	i1ProTankPumpLPM : INT; (* Byte "n+100, n+101" *)
	i2ProTankPumpHz : INT; (* Byte "n+102, n+103" *)
	i3ProTankBtmUsAPwrPercent : INT; (* Byte "n+104, n+105" *)
	i4ProTankBtmUsBPwrPercent : INT; (* Byte "n+106, n+107" *)
	i5ProTankBtmUsCPwrPercent : INT; (* Byte "n+108, n+109" *)
	i6ProTankSideUsAPwrPercent : INT; (* Byte "n+110, n+111" *)
	i7ProTankSideUsBPwrPercent : INT; (* Byte "n+112, n+113" *)
	i8ProTankBtmUsAkHz : INT; (* Byte "n+114, n+115" *)
	i9ProTankBtmUsBkHz : INT; (* Byte "n+116, n+117" *)
	i10ProTankBtmUsCkHz : INT; (* Byte "n+118, n+119" *)
	i11ProTankSideUsAkHz : INT; (* Byte "n+120, n+121" *)
	i12ProTankSideUsBkHz : INT; (* Byte "n+122, n+123" *)
	i13ProTankBlowerHz : INT; (* Byte "n+124, n+125" *)
	r14ProTankChangeTempDegC : REAL; (*Byte " n+126, n+129" *) (*New*)
	r15SubTankChangeTempDegC :REAL; (*Byte "N+130, n+133" *) (*New*)
	i16SubTankPumpLPM : INT; (*Byte "N+134, n+135" *) (*New*)
	i17SubTankPumpHz : INT; (*Byte "N+136, n+137" *) (*New*)
	i18SlowPullVelocity   : INT;(* Byte "n+154, n+155" *) (*MODIFIED*)
	i19SlowPullDelayTime   : INT;(* Byte "n+154, n+155" *) (*MODIFIED*)


	sReservedInt : STRING(50); (* Byte "n+138~n+199" *)





END_STRUCT
END_TYPE

// ---- DUTs/DS TBD/DS_SubRecipeMemory.TcDUT
TYPE DS_SubRecipeMemory : (*Full Occupied Byte = 400*)
STRUCT
(*BOOL - Start Condition*)
(*	bStCon1EnLowLiquidLevel : BOOL; (* Byte "n" *)
	bStCon2EnRegLiquidLevel : BOOL; (* Byte "n+1" *)
	bStCon3EnLowVacuumLevel : BOOL; (* Byte "n+2" *)
	bStCon4EnRegVacuumLevel : BOOL; (* Byte "n+3" *)
	bStCon5EnLowPressureLevel : BOOL; (* Byte "n+4" *)
	bStCon6EnRegPressureLevel : BOOL; (* Byte "n+5" *)
	bStCon7EnBelowTargetVacuumLevel : BOOL; (* Byte "n+6" *)
	bStCon8EnAboveTargetVacuumLevel : BOOL; (* Byte "n+7" *)
	bStCon9EnBelowTargetPressureLevel : BOOL; (* Byte "n+8" *)
	bStCon10EnAboveTargetPressureLevel : BOOL; (* Byte "n+9" *)
	bStCon11EnBelowTargetProTankTempLevel : BOOL; (* Byte "n+10" *)
	bStCon12EnAboveTargetProTankTempLevel : BOOL; (* Byte "n+11" *)
	bStCon13EnBelowTargetSubTankTempLevel : BOOL; (* Byte "n+12" *)
	bStCon14EnAboveTargetSubTankTempLevel : BOOL; (* Byte "n+13" *)
	bStCon15ExternalActivation : BOOL; (* Byte "n+14" *)
*)
	bStCon1EnProLowLiquidLevel : BOOL; (* Byte "n" *)
	bStCon2EnProRegLiquidLevel : BOOL; (* Byte "n+1" *)
	bStCon3EnProHighLiquidLevel : BOOL; (* Byte "n+1" *)

	bStCon4EnSubLowLiquidLevel : BOOL; (* Byte "n+1" *)
	bStCon5EnSubRegLiquidLevel : BOOL; (* Byte "n+1" *)
	bStCon6EnSubHighLiquidLevel : BOOL; (* Byte "n+1" *)

	bStCon7EnLowVacuumLevel : BOOL; (* Byte "n+2" *)
	bStCon8EnRegVacuumLevel : BOOL; (* Byte "n+3" *)
	bStCon9EnLowPressureLevel : BOOL; (* Byte "n+4" *)
	bStCon10EnRegPressureLevel : BOOL; (* Byte "n+5" *)
	bStCon11EnBelowTargetVacuumLevel : BOOL; (* Byte "n+6" *)
	bStCon12EnAboveTargetVacuumLevel : BOOL; (* Byte "n+7" *)
	bStCon13EnBelowTargetPressureLevel : BOOL; (* Byte "n+8" *)
	bStCon14EnAboveTargetPressureLevel : BOOL; (* Byte "n+9" *)
	bStCon15EnBelowTargetProTankTempLevel : BOOL; (* Byte "n+10" *)
	bStCon16EnAboveTargetProTankTempLevel : BOOL; (* Byte "n+11" *)
	bStCon17EnBelowTargetSubTankTempLevel : BOOL; (* Byte "n+12" *)
	bStCon18EnAboveTargetSubTankTempLevel : BOOL; (* Byte "n+13" *)
	bStCon19ExternalActivation : BOOL; (* Byte "n+14" *)

(*BOOL - Complete Condition*)
	bComCon1EnProLowLiquidLevel : BOOL; (* Byte "n+15" *)
	bComCon2EnProRegLiquidLevel : BOOL; (* Byte "n+16" *)
	bComCon3EnProHighLiquidLevel : BOOL; (* Byte "n+16" *)

	bComCon4EnSubLowLiquidLevel : BOOL; (* Byte "n+16" *)
	bComCon5EnSubRegLiquidLevel : BOOL; (* Byte "n+16" *)
	bComCon6EnSubHighLiquidLevel : BOOL; (* Byte "n+16" *)

	bComCon7EnLowVacuumLevel : BOOL; (* Byte "n+17" *)
	bComCon8EnRegVacuumLevel : BOOL; (* Byte "n+18" *)
	bComCon9EnLowPressureLevel : BOOL; (* Byte "n+19" *)
	bComCon10EnRegPressureLevel : BOOL; (* Byte "n+20" *)
	bComCon11EnBelowTargetVacuumLevel : BOOL; (* Byte "n+21" *)
	bComCon12EnAboveTargetVacuumLevel : BOOL; (* Byte "n+22" *)
	bComCon13EnBelowTargetPressureLevel : BOOL; (* Byte "n+23" *)
	bComCon14EnAboveTargetPressureLevel : BOOL; (* Byte "n+24" *)
	bComCon15EnBelowTargetProTankTempLevel : BOOL; (* Byte "n+25" *)
	bComCon16EnAboveTargetProTankTempLevel : BOOL; (* Byte "n+26" *)
	bComCon17EnBelowTargetSubTankTempLevel : BOOL; (* Byte "n+27" *)
	bComCon18EnAboveTargetSubTankTempLevel : BOOL; (* Byte "n+28" *)
	bComCon19EnExternalActivation : BOOL; (* Byte "n+29" *)
	bComCon20EnProcessTimer : BOOL; (* Byte "n+29" *)

(*BOOL - Instrument Output*)
	bOut1EnProTankPump : BOOL; (* Byte "n+30" *)
	bOut2EnProTankHeater : BOOL; (* Byte "n+31" *)
	bOut3EnProTankBottomUltrasonicA : BOOL; (* Byte "n+32" *)
	bOut4EnProTankBottomUltrasonicB : BOOL; (* Byte "n+33" *)
	bOut5EnProTankBottomUltrasonicC : BOOL; (* Byte "n+34" *)
	bOut6EnProTankSideUltrasonicA : BOOL; (* Byte "n+35" *)
	bOut7EnProTankSideUltrasonicB : BOOL; (* Byte "n+36" *)
	bOut8EnSubTankPump : BOOL; (* Byte "n+37" *)
	bOut9EnSubTankHeater : BOOL; (* Byte "n+38" *)
	bOut10EnBlower : BOOL; (* Byte "n+39" *)
	bOut11EnVacuumPump : BOOL; (* Byte "n+40" *)
	bOut12EnSlowPull : BOOL; (* Byte "n+41" *) (*MODIFIED*)
	bOut13EnInstrument2 : BOOL; (* Byte "n+42" *)
	bOut14EnInstrument3 : BOOL; (* Byte "n+43" *)
	bOut15EnInstrument4 : BOOL; (* Byte "n+44" *)

(*BOOL - Valve Output*)
	bOut1ActValve1 : BOOL; (* Byte "n+45" *)
	bOut2ActValve2 : BOOL; (* Byte "n+46" *)
	bOut3ActValve3 : BOOL; (* Byte "n+47" *)
	bOut4ActValve4 : BOOL; (* Byte "n+48" *)
	bOut5ActValve5 : BOOL; (* Byte "n+49" *)
	bOut6ActValve6 : BOOL; (* Byte "n+50" *)
	bOut7ActValve7 : BOOL; (* Byte "n+51" *)
	bOut8ActValve8 : BOOL; (* Byte "n+52" *)
	bOut9ActValve9 : BOOL; (* Byte "n+53" *)
	bOut10ActValve10 : BOOL; (* Byte "n+54" *)
	bOut11ActValve11 : BOOL; (* Byte "n+55" *)
	bOut12ActValve12 : BOOL; (* Byte "n+56" *)
	bOut13ActValve13 : BOOL; (* Byte "n+57" *)
	bOut14ActValve14 : BOOL; (* Byte "n+58" *)
	bOut15ActValve15 : BOOL; (* Byte "n+59" *)
	bOut16ActValve16 : BOOL; (* Byte "n+60" *)
	bOut17ActValve17 : BOOL; (* Byte "n+61" *)
	bOut18ActValve18 : BOOL; (* Byte "n+62" *)
	bOut19ActValve19 : BOOL; (* Byte "n+63" *)
	bOut20ActValve20 : BOOL; (* Byte "n+64" *)


(*BOOL - Instrument Output*) (*New*)
	bOut16EnProTankChangeTemperature : BOOL; (* Byte "n+65" *) (*New*)
	bOut17EnSubTankChangeTemperature : BOOL; (* Byte "n+66" *) (*New*)


	sReservedBool : STRING(50); (* Byte "n+67~n+99" *)


(*INT - Start Condition*)

	iStCon1TargetVacuumLevel : INT; (* Byte "n+100, n+101" *)
	iStCon2TargetPressureLevel : INT; (* Byte "n+102, n+103" *)
	iStCon3TargetProTankTempLevel : INT; (* Byte "n+104, n+105" *)
	iStCon4TargetSubTankTempLevel : INT; (* Byte "n+106, n+107" *)

(*INT - Complete Condition*)

	iComCon1TargetVacuumLevel : INT; (* Byte "n+108, n+109" *)
	iComCon2TargetPressureLevel : INT; (* Byte "n+110, n+111" *)
	iComCon3TargetProTankTempLevel : INT; (* Byte "n+112, n+113" *)
	iComCon4TargetSubTankTempLevel : INT; (* Byte "n+114, n+115" *)
	iComCon5ProcessTimer : INT; (* Byte "n+116, n+117" *)

(*INT - Power/Flow Control*)
	iOut1ProTankPumpLPM : INT; (* Byte "n+118, n+119" *)
	iOut2ProTankPumpHz : INT; (* Byte "n+120, n+121" *)
	iOut3ProTankBtmUsAPwrPercent : INT; (* Byte "n+122, n+123" *)
	iOut4ProTankBtmUsBPwrPercent : INT; (* Byte "n+124, n+125" *)
	iOut5ProTankBtmUsCPwrPercent : INT; (* Byte "n+126, n+127" *)
	iOut6ProTankSideUsAPwrPercent : INT; (* Byte "n+128, n+129" *)
	iOut7ProTankSideUsBPwrPercent : INT; (* Byte "n+130, n+131" *)
	iOut8ProTankBtmUsAkHz : INT; (* Byte "n+132, n+133" *)
	iOut9ProTankBtmUsBkHz : INT; (* Byte "n+134, n+135" *)
	iOut10ProTankBtmUsCkHz : INT; (* Byte "n+136, n+137" *)
	iOut11ProTankSideUsAkHz : INT; (* Byte "n+138, n+139" *)
	iOut12ProTankSideUsBkHz : INT; (* Byte "n+140, n+141" *)
	iOut13ProTankBlowerHz : INT;(* Byte "n+142, n+143" *)

	rOut14ProTankChangeTemperatureDegC  : REAL;(* Byte "n+144, n+147" *) (*New*)
	rOut15SubTankChangeTemperatureDegC  : REAL;(* Byte "n+148, n+151" *) (*New*)
	iOut16SubTankPumpLPM   : INT;(* Byte "n+152, n+153" *) (*New*)
	iOut17SubTankPumpHz   : INT;(* Byte "n+154, n+155" *) (*New*)

	iOut18SlowPullVelocity   : INT;(* Byte "n+154, n+155" *) (*MODIFIED*)
	iOut19SlowPullDelayTime   : INT;(* Byte "n+154, n+155" *) (*MODIFIED*)



	sReservedInt : STRING(50); (* Byte "n+156~n+159" *)


(*LREAL - Standby*)
	lrLREALReserved1 : LREAL; (* Byte "n+160~n+167" *)
	lrLREALReserved2 : LREAL; (* Byte "n+168~n+175" *)
	sReservedLreal : STRING(50); (* Byte "n+176~n+199" *)


(*STRING - Standby*)
	sStringReserved1 : STRING(50); (* Byte "n+200 ~ n+299" *)
	sStringReserved2 : STRING(50); (* Byte "n+300 ~ n+399" *)







END_STRUCT
END_TYPE

// ---- DUTs/DS TBD/DS_TimeTrackerInput.TcDUT
TYPE DS_TimeTrackerInput :
STRUCT
(* from DSA1_PnpSequenceMemory*)

(*	bTimeTrackerEn : BOOL;*)
	iTimeTrackerProductRecipeNo : INT;
(*	iTimeTrackerStepNo : INT; (*Byte "n+110, n+111" *) (***************NEW******************)*)

	ARiCallArmNo : ARRAY [0..iProductRecipeStepArrayQty] OF INT; (* Byte "n+100~n+161" *)

	ARiPickStationNo : ARRAY [0..iProductRecipeStepArrayQty] OF INT; (* Byte "n+162~n+223" *)
	ARiTransferStationNo : ARRAY [0..iProductRecipeStepArrayQty] OF INT; (* Byte "n+224~n+285" *)

	ARiStnSeqRepNo : ARRAY [0..iProductRecipeStepArrayQty] OF INT; (* Byte "n+596~n+657" *)

END_STRUCT

END_TYPE

// ---- DUTs/DS TBD/DS_WeberEnclosure.TcDUT
TYPE DS_WeberEnclosure :
STRUCT
	DSWeberGenerator : ARRAY [1..iUSGeneratorQty] OF DS_WeberGenerator;
END_STRUCT
END_TYPE

// ---- DUTs/DS TBD/DS_WeberGenerator.TcDUT
TYPE DS_WeberGenerator :
STRUCT
	IN_bUltrasonicStartEn : BOOL;
	IN_bMultiFreqEn :  BOOL;
	IN_iFreqSetPoint :  INT; (* 40/80/120 or 25/50*)
	IN_iTargetPowerPercentSetPoint :  INT; (* 0-100%*)
	IN_lrPowerToAnalogRatio : LREAL; (*Normally for 0-100% is 327.67*)
	IN_lrAnalogInputFineTuneRatio :  LREAL; (*Normally 1, use lower than 1 (example: 0.97) if set to 100% the actual output is greater, use higher than 1 meant the actual output is lesser when you set 100% *)
	IN_lrAnalogOutputFineTuneRatio :  LREAL; (*Normally 1, use lower than 1 (example: 0.97) if set to 100% the actual output is greater, use higher than 1 meant the actual output is lesser when you set 100% *)

	DSWeberMulFreqSwitching : DS_WeberMulFreqSwitching;

	OUT_bUltrasonicOnOff :  BOOL;
	OUT_iActualPowerPercentDisplay :  INT; (*Display 0 - 100%*)
	OUT_bFreqSetPointError :  BOOL;

	IN_iPowerAnalogInput  :  INT; (*Link to Terminal*)
	OUT_iPowerAnalogOutput  :  INT; (*Link to Terminal*)

END_STRUCT
END_TYPE

// ---- DUTs/DS TBD/DS_WeberMulFreqSwitching.TcDUT
TYPE DS_WeberMulFreqSwitching :
STRUCT
	bFreqSwitchingPB_TS : BOOL;
	bFreqRange4080120En : BOOL;
	bFreqRange2550En : BOOL;
	bDisableMultiFreq80kHz : BOOL;
	bDisableMultiFreq40kHz : BOOL;
	iFreqOutput_TS : INT;
END_STRUCT
END_TYPE

// ---- DUTs/DS TBD/DS_XMLRW.TcDUT
TYPE DS_XMLRW :
STRUCT

	sMachineOnTime_JKS	: STRING(99);

END_STRUCT
END_TYPE

// ---- DUTs/DS TBD/DS_XML_InputOutput.TcDUT
TYPE DS_XML_InputOutput :
STRUCT

(*	var1									: ARRAY [1..iStnQty] OF BOOL;
	ARrStnTempSV_map					: ARRAY [1..iStnQty] OF REAL;
	ARrStnTempPV_map					: ARRAY [1..iStnQty] OF REAL;
	ARrStnTempHALsv_map				: ARRAY [1..iStnQty] OF REAL;
	ARrStnTempRDYsv_map				: ARRAY [1..iStnQty] OF REAL;
	ARrStnTempHYSsv_map				: ARRAY [1..iStnQty] OF REAL;
	ARrStnTemp1stLimitSv_map			: ARRAY [1..iStnQty] OF REAL;
	ARiStnPreparationTempSv_map		: ARRAY [1..iStnQty] OF INT;

	ARrStnSubTankTempSV_map			: ARRAY [1..iStnQty] OF REAL;
	ARrStnSubTankTempPV_map			: ARRAY [1..iStnQty] OF REAL;
	ARrStnSubTankTempHALsv_map		: ARRAY [1..iStnQty] OF REAL;
	ARrStnSubTankTempRDYsv_map		: ARRAY [1..iStnQty] OF REAL;
	ARrStnSubTankTempHYSsv_map		: ARRAY [1..iStnQty] OF REAL;
	ARrStnSubTankTemp1stLimitSv_map	: ARRAY [1..iStnQty] OF REAL;
	ARiStnSubTankPreparationTempSv_map: ARRAY [1..iStnQty] OF INT;


	ARiStnDippingTimeSV_map			: ARRAY [1..iStnQty] OF INT;
	ARiStnToleranceTimeSV_map			: ARRAY [0..iStnQty] OF INT;
	ARiStnTopUpDelayOffTimeSV_map		: ARRAY [1..iStnQty] OF INT;
*)
	ARrStnConductivityPV_map 			: ARRAY [1..iStnQty] OF REAL;
	ARrStnConductivity1stLimitSv_map		: ARRAY [1..iStnQty] OF REAL;
	ARrStnConductivity2ndLimitSv_map		: ARRAY [1..iStnQty] OF REAL;
(*
	ARrStnPhPV_map						: ARRAY [1..iStnQty] OF REAL;
	ARrStnLowPHSv_map					: ARRAY [1..iStnQty] OF REAL;
	ARrStnHighPHSv_map					: ARRAY [1..iStnQty] OF REAL;

	ARrStnFilterPressurePV_map 			: ARRAY [1..iStnQty] OF REAL;
	ARrStnLowFilterPressureSv_map		: ARRAY [1..iStnQty] OF REAL;
	ARrStnHighFilterPressureSv_map		: ARRAY [1..iStnQty] OF REAL;
*)
END_STRUCT
END_TYPE

// ---- DUTs/DS TBD/En_LogFileType.TcDUT
TYPE En_LogFileType :
(
	CSV:=1,
	TXT:=2
);
END_TYPE

// ---- DUTs/DS TBD/En_TimeInterval.TcDUT
TYPE En_TimeInterval :
(
	Interval_1s:=12,
	Interval_5s:=13,
	Interval_10s:=0,
	Interval_20s:=1,
	Interval_30s:=2,
	Interval_1min:=3,
	Interval_2min:=4,
	Interval_5min:=5,
	Interval_10min:=6,
	Interval_15min:=7,
	Interval_20min:=8,
	Interval_30min:=9,
	Interval_1h:=10,
	Interval_2h:=11

);
END_TYPE

// ---- DUTs/DS Twincat 3/Barcode/DS_SerialCommunication.TcDUT
TYPE DS_SerialCommunication :
STRUCT
	// Config
	SerialCfg 				: ComSerialConfig;
	PortOpened 				: BOOL;     (* Indicates if selected serial port is opened *)
    SerialConnectError      : BOOL;     (* 'TRUE' if an error occurred *)
    ErrorID    				: UDINT;    (* Displays the error code; 0 = no error *)
    Busy       				: BOOL;     (* 'TRUE' if internal ADS communication is busy *)
    TxBufCount 				: UDINT;    (* number of bytes in internal Tx buffer *)
    RxBufCount 				: UDINT;    (* number of bytes in internal Rx buffer *)	
    Error 					: BOOL;
	RxTimeout 				: BOOL;
	StringReceived 			: BOOL;
	TxBuffer				: ComBuffer;
	RxBuffer				: ComBuffer;

	// Send String Input
	sSendString 			: STRING;
	bSendStringBusy 		: BOOL;
	SendStringError 		: ComError_t;
	
	// Receive String Input//
	sReceivedString 		: STRING;
	bStringReceived			: BOOL;
	ReceivedStringError 	: ComError_t;
	bReceivedStringBusy 	: BOOL;
	bReceivedStringTimeout	: BOOL;
	bReceivedStringReset	: BOOL;	
	sRSPrefix 				: STRING;
    sRSSuffix 				: STRING;
	
END_STRUCT
END_TYPE

// ---- DUTs/DS Twincat 3/CSV/DS_CsvErrorLog.TcDUT
TYPE DS_CsvErrorLog EXTENDS DS_CsvLog :
STRUCT
	udiErrorId	: UDINT;
	iCaseid		: INT;
END_STRUCT
END_TYPE

// ---- DUTs/DS Twincat 3/CSV/DS_CsvLog.TcDUT
TYPE DS_CsvLog :
STRUCT
		eLogAction			: E_CsvActionType; 
		sPathAndFilename	: STRING(255);
		sLogString			: STRING(255);
END_STRUCT
END_TYPE

// ---- DUTs/DS Twincat 3/CSV/DS_CsvReport.TcDUT
TYPE DS_CsvReport :
STRUCT
	
	ARsHeadlineTitle			: ARRAY [1..100] OF STRING;		// Please consider to replace the name on next project
	ARsHeadlineData				: ARRAY [1..100] OF STRING;	                		
	ARsLogUnit					: ARRAY [1..100] OF STRING;
	ARsLogTitle					: ARRAY [1..100] OF STRING;
	AR2sLogData					: ARRAY [1..100]OF ARRAY [1..C_iCsvDataBlockQty] OF STRING;

	iNumOfData_HeadlineTitle 	: INT := 50;
	iNumOfData_HeadlineData		: INT := 50;
	iNumOfData_LogUnit			: INT := 50;
	iNumOfData_LogTitle			: INT := 50;
	iNumOfData_LogData			: INT := 50;

	ARsLogTitle_EventLog 			: ARRAY [1..C_iCsvDataBlockQty] OF STRING;
	ARsLogData_EventLog 			: ARRAY [1..C_iCsvDataBlockQty] OF STRING;

	iNumOfData_LogTitle_EventLog 	: INT := 10;
	iNumOfData_LogData_EventLog 	: INT := 10;
	
	ARsLogBuffer		: ARRAY [1..C_udiCsvBufferByteQty] OF BYTE; 
	
END_STRUCT
END_TYPE

// ---- DUTs/DS Twincat 3/CSV/E_CsvActionType.TcDUT
{attribute 'Tc2GvlVarNames'}
{attribute 'strict'}
{attribute 'to_String'}
TYPE E_CsvActionType :
(
	eCsvNewFile_CarrierReport 	:= 1,
	eCsvLogData_CarrierReport	:= 2,
	eCsvGenerate_CarrierReport	:= 3,
	eCsvNewFile_EventLog 		:= 4,
	eCsvLogData_EventLog		:= 5,
	eCsvGenerate_EventLog		:= 6
	
);
END_TYPE

// ---- DUTs/DS Twincat 3/DS_HMI_MappingVariable.TcDUT
TYPE DS_HMI_MappingVariable :
STRUCT
	
//PushButton

bProTankHeater_PB				:BOOL;
bProTankPump_PB				    :Bool;
bProTankUsSide_PB				:Bool;
bProTankUsBtm_PB				:Bool;
bProTankUsFreqChangeBit1_PB	    :Bool;
bProTankUsFreqChangeBit2_PB     :Bool;
bProTankVacuumPump_PB			:Bool;
bProTankAgitationMotor_PB		:BOOL;
bProTankBlower_PB				:BOOL;
bDosingPump_PB				    :BOOL;
bLdConveyorMotor01_PB			:BOOL;
bLdConveyorMotor02_PB			:BOOL;
bLdConveyorMotor03_PB			:BOOL;
bLdConveyorMotor04_PB			:BOOL;
bValve01_PB					    :BOOL;
bValve02_PB					    :Bool;
bValve03_PB					    :Bool;
bValve04_PB					    :Bool;
bValve05_PB					    :BOOL;
bExhaustBlower_PB				:BOOL;
bStnRotationRotaryBarrel_PB		:BOOL;
bRobotRotationRotaryBarrel_PB   :BOOL;
bGeneralIncValve01_PB 			:BOOL;
bGeneralIncValve02_PB 			:BOOL;
bFFU01_PB				 		:BOOL;
bFFU02_PB				 		:BOOL;




//Indicator
bProTankHeater_IND				:BOOL;
bProTankPump_IND	  			:BOOL;
bProTankUsSide_IND				:BOOL;
bProTankUsBtm_IND				:BOOL;
bProTankUsFreqChangeBit1_IND	:BOOL;
bProTankUsFreqChangeBit2_IND    :BOOL;
bProTankVacuumPump_IND			:BOOL;
bProTankAgitationMotor_IND		:BOOL;
bProTankBlower_IND				:BOOL;
bDosingPump_IND	    			:BOOL;
bLdConveyorMotor01_IND			:BOOL;
bLdConveyorMotor02_IND			:BOOL;
bLdConveyorMotor03_IND			:BOOL;
bLdConveyorMotor04_IND			:BOOL;
bValve01_IND			  		:BOOL;
bValve02_IND			  		:BOOL;
bValve03_IND			  		:BOOL;
bValve04_IND			  		:BOOL;
bValve05_IND			  		:BOOL;
bExhaustBlower_IND				:BOOL;
bStnRotationRotaryBarrel_IND	:BOOL;
bRobotRotationRotaryBarrel_IND  :BOOL;
bGeneralIncValve01_IND 			:BOOL;
bGeneralIncValve02_IND 			:BOOL;


bProcessTankMinLevel_IND		:BOOL;
bProcessTankRegLevel_IND		:BOOL;
bProcessTankTopupLevel_IND		:BOOL;

bSubTankMinLevel_IND			:BOOL;
bSubTankRegLevel_IND			:BOOL;
bSubTankMaxLevel_IND			:BOOL;
bSubTankTopupLevel_IND			:BOOL;

bOverflowMinLevel_IND			:BOOL;
bOverflowRegLevel_IND			:BOOL;
bOverflowMaxLevel_IND			:BOOL;

bLdFeedSensor_IND				:BOOL;
bLdIndex1Sensor_IND				:BOOL;
bLdIndex2Sensor_IND				:BOOL;
bLdIndex3Sensor_IND				:BOOL;
bLdIndex4Sensor_IND				:BOOL;
bLdPickSensor_IND				:BOOL;

bUldFeedSensor_IND				:BOOL;
bUldIndex1Sensor_IND			:BOOL;
bUldIndex2Sensor_IND			:BOOL;
bUldIndex3Sensor_IND			:BOOL;
bUldIndex4Sensor_IND			:BOOL;
bUldPickSensor_IND				:BOOL;

bFFU01_IND				 		:BOOL;
bFFU02_IND				 		:BOOL;




END_STRUCT
END_TYPE

// ---- DUTs/DS Twincat 3/DS_LocalSystemTime.TcDUT
TYPE DS_LocalSystemTime :
STRUCT

dtCurrentDateTime			: DT; 		  // Newly Added DT#2023-02-20-15:49:44
sCurrentDateTime			: STRING(30); // Newly Added 2023-02-20-15:49:44
sCurrentDate_General		: STRING(255); // Newly Added YYYYMMDD
sCurrentTime24Hr_General	: STRING(50); // Newly Added HH:MM:SS	
sCurrentDT24Hr_General		: STRING(50);
sCurrentDT12Hr				: STRING(50);
sCurrentDT24Hr				: STRING(50);
sDayOfWeek					: STRING(10);
sYear						: STRING(10);
sMonth						: STRING(10);
sDay						: STRING(10);
s24Hour						: STRING(10);
s12Hour						: STRING(10);
sMin						: STRING(10);
sSec						: STRING(10);
s12HrSign					: STRING(10);

END_STRUCT
END_TYPE

// ---- DUTs/DS Twincat 3/DS_XML_Persistent_Analog.TcDUT
TYPE DS_XML_Persistent_Analog :
STRUCT
	(* xxxxxxxxxxxxxxxxxxxxxxxxxxxxxxxx Temperature Cltr xxxxxxxxxxxxxxxxxxxxxxxxxxxxxxxx*)
(*========================================================================*)

	ARfbStnTempControl									: ARRAY [1..iStnQty] OF fbV2_TempControl;

	ARrAnalogInputFineTuneRatio							: ARRAY [1..iStnQty] OF REAL;

	ARrStnTempHYSsv										: ARRAY [1..iStnQty] OF REAL;
	ARrStnTempHALsv										: ARRAY [1..iStnQty] OF REAL;
	ARrStnTempSV										: ARRAY [1..iStnQty] OF REAL;
	ARrStnTempRDYsv										: ARRAY [1..iStnQty] OF REAL;
	ARrStnTemp1stLimitSv								: ARRAY [1..iStnQty] OF REAL;
	ARrStnTemp2ndLimitSv								: ARRAY [1..iStnQty] OF REAL;
	ARiStnPreparationTempSv								: ARRAY [1..iStnQty] OF INT;
	
	fbChillerSystemTempControl							: fbV2_TempControl;
	
	rChillerSystemAnalogInputFineTuneRatio				: REAL;

	rChillerSystemTempHYSsv								: REAL;
	rChillerSystemTempHALsv								: REAL;
	rChillerSystemTempSV								: REAL;
	rChillerSystemTempRDYsv								: REAL;
	rChillerSystemTemp1stLimitSv						: REAL;
	rChillerSystemTemp2ndLimitSv						: REAL;
	iChillerSystemPreparationTempSv						: INT;

	ARrStnChillerValueTempSetpoint						: ARRAY [1..iStnQty] OF REAL;
	
(*****Temperature Changed Based on Recipe Ctrl *****)

	fbTemperatureParaRecipe								: fbV3_TemperatureParaRecipe;

	DSTempCtrlParameter_Min 							: DSV3_TempCtrlParameter;
	DSTempCtrlParameter_Max 							: DSV3_TempCtrlParameter;

	HMI_DSTempCtrlParameter_Input 						: DSV3_TempCtrlParameter;

(* xxxxxxxxxxxxxxxxxxxxxxxxxxxxxxxx Conductivity Cltr xxxxxxxxxxxxxxxxxxxxxxxxxxxxxxxx*)
(*========================================================================*)

	ARfbStnConductivity 								: ARRAY [1..iStnQty] OF fbRawRatioConversionReal;

	ARrStnLowConductivitySv								: ARRAY [1..iStnQty] OF REAL;
	ARrStnHighConductivitySv							: ARRAY [1..iStnQty] OF REAL;
	ARrStnConductivity1stLimitSv						: ARRAY [1..iStnQty] OF REAL;
	ARrStnConductivity2ndLimitSv						: ARRAY [1..iStnQty] OF REAL;

	bStnConductivityMaxLimitReach						: ARRAY [1..iStnQty] OF BOOL;
	ARsConductivityMsgStatus							: ARRAY [1..iStnQty] OF STRING;

(* xxxxxxxxxxxxxxxxxxxxxxxxxxxxxxxx Filter Pressure Cltr xxxxxxxxxxxxxxxxxxxxxxxxxxxxxxxx*)
(*========================================================================*)

	ARfbStnFilterPressure 								: ARRAY [1..iStnQty] OF fbRawRatioConversionReal;
                                                    
	ARrStnLowFilterPressureSv							: ARRAY [1..iStnQty] OF REAL;
	ARrStnHighFilterPressureSv							: ARRAY [1..iStnQty] OF REAL;
	ARrStnFilterPressure1stLimitSv						: ARRAY [1..iStnQty] OF REAL;
	ARrStnFilterPressure2ndLimitSv						: ARRAY [1..iStnQty] OF REAL;
                                                    
	ARfbIncFilterPressure								: ARRAY [1..iStnQty] OF fbRawRatioConversionReal;
	ARrIncLowFilterPressureSv							: ARRAY [1..iStnQty] OF REAL;
	ARrIncHighFilterPressureSv							: ARRAY [1..iStnQty] OF REAL;
	ARrIncFilterPressure1stLimitSv						: ARRAY [1..iStnQty] OF REAL;
	ARrIncFilterPressure2ndLimitSv						: ARRAY [1..iStnQty] OF REAL;


(* xxxxxxxxxxxxxxxxxxxxxxxxxxxx Clangsonic Ultrasonic Cltr xxxxxxxxxxxxxxxxxxxxxxxxxxxx*)
(*========================================================================*)

	DSClangGenerator 									: ARRAY [1..iUSGeneratorQty] OF DS_ClangsonicGenerator;
	DSClangGenerator2 									: ARRAY [1..iUSGeneratorQty] OF DS_ClangsonicGenerator;
	iClangStepDelaySVns									: INT := 50;
	iClangStepDelaySVns2								: INT := 50;

	iClangTolerance										: INT;
	iUSTolerance										: INT;
	ARlrUsMaxData_Watt									: ARRAY [1..12] OF LREAL;

	DSClangsonicGenerator 								: DSV2_ClangsonicGenerator;
	DSClangsonicGenerator2 								: DSV2_ClangsonicGenerator;

	
(* xxxxxxxxxxxxxxxxxxxxxxxxxxx Modbus Cltr xxxxxxxxxxxxxxxxxxxxxxxxxxx*)
(*========================================================================*)
	DSV2ModbusControl									: DSV2_ModbusControl;
	DSV2ModbusControl2 									: DSV2_ModbusControl;
	
	IStepDelaySVns										: INT := 50;
	IStepDelaySVns2										: INT := 50;


END_STRUCT
END_TYPE

// ---- DUTs/DS Twincat 3/DS_XML_Persistent_Arm.TcDUT
TYPE DS_XML_Persistent_Arm :
STRUCT
	(* xxxxxxxxxxxxxxxxxxxxxxxxxxxxxxxxxxx  Station Info xxxxxxxxxxxxxxxxxxxxxxxxxxxxxxxxxxx*)
(*========================================================================*)

	bEnableCallArmNo 						: BOOL;
	iCallArmNo 								: INT;
	ARiVertArmPosOffset 					: ARRAY [0..iArmQty] OF INT;

	bAgitationEn							: BOOL;
	bArm2AgitationEn						: BOOL;
(* xxxxxxxxxxxxxxxxxxxxxxxxxxx  Display Product Description xxxxxxxxxxxxxxxxxxxxxxxxxxx*)
(*========================================================================*)

	ARsProductRecipeDescription				: ARRAY [0..iProductRecipeArrayQty] OF STRING(50);
	DSHmiStationDisplayInfo 				: ARRAY [1..iStnQty] OF DS_HMIStationDisplayInfo;

	ARbStnSeqRepNoVisible					: ARRAY [0..iProductRecipeStepArrayQty] OF BOOL;
	ARsStnProcessStatus 					: ARRAY [0..iStnQty] OF STRING;

(* xxxxxxxxxxxxxxxxxxxxxx  Arm PnP Sequence Memory Description xxxxxxxxxxxxxxxxxxxxxx*)
(*========================================================================*)

	DSA1fbPnpSequenceMemoryCall 			: DSV2_A1_fbPnpSequenceMemoryCall;
	DSA1fbPnpSequenceMemoryStore 			: DSV2_A1_fbPnpSequenceMemoryStore;
	DSA21UpDownPatternCall 					: DSA21_UpDownPatternCall;
	DSA21UpDownPatternStore 				: DSA21_UpDownPatternStore;
	DSA31ArmSpeedProfileCall 				: DSA31_ArmSpeedProfileCall;
	DSA31ArmSpeedProfileStore 				: DSA31_ArmSpeedProfileStore;

(* xxxxxxxxxxxxxxxxxxxxxxxxxxxxx Admin Arm Setting xxxxxxxxxxxxxxxxxxxxxxxxxxxxxxxxxxxxxxx*)
(*========================================================================*)

	DSHomingSetting 						: DS_HomingSetting;

	ARDSArmCtrl 							: ARRAY [0..iArmQty] OF DSV2_ArmPosition;
	(*1 = Stn, 2 = Id, 3 = Uld*)
	(*1 = Up, 2 = SPSlanted, 3 = Regular(*midtop*), 4 = AgitationUp, 5 = AgitationDown, 6 = Down, 7 = Unhook, 8 = Hook, 9 = SlantedLeft, 10 = SlantedRight
		,11 = lifter up, 12 = lifter = down*)

(* xxxxxxxxxxxxxxxxxxxxx  4 Step Arm Movement - Auto/Manual Used xxxxxxxxxxxxxxxxxxxxxxxxxx*)
(*==============================================================================*)

	DS4StepsMovement 						: DS_SA_Movement;
	DSManual4StepsMovement					: DS_SA_Movement;


(* xxxxxxxxxxxxxxxxxxxxxxxxxxx Arm 1 Vert / Horz Velo,Acc,Dcc xxxxxxxxxxxxxxxxxxxxxxxxxxx*)
(*========================================================================*)

	ARlrArmVertFix_PosCfmTolerance			: ARRAY [0..iArmQty] OF LREAL;
	ARlrArmVertFix_2ndSpdRange				: ARRAY [0..iArmQty] OF LREAL;

	ARlrArmHorzFix_PosCfmTolerance			: ARRAY [0..iArmQty] OF LREAL;
	ARlrArmHorzFix_2ndSpdRange				: ARRAY [0..iArmQty] OF LREAL;

(* xxxxxxxxxxxxxxxxxxxxxxxxxxxxxxx Jog Control Variable xxxxxxxxxxxxxxxxxxxxxxxxxxxxxxxxxxxxx*)
(*============================================================================*)

	ARrArmVertJogPercent					: ARRAY [1..iArmQty] OF REAL;
	ARrArmVertJogAcc						: ARRAY [1..iArmQty] OF REAL;
	ARrArmVertJogDcc						: ARRAY [1..iArmQty] OF REAL;

	ARrArmHorzJogPercent					: ARRAY [1..iArmQty] OF REAL;
	ARrArmHorzJogAcc						: ARRAY [1..iArmQty] OF REAL;
	ARrArmHorzJogDcc						: ARRAY [1..iArmQty] OF REAL;

	ARlrArmSlowPullJogVelo					: ARRAY [1..iArmSlowPullQty] OF LREAL;
	ARlrArmSlowPullJogAcc					: ARRAY [1..iArmSlowPullQty] OF LREAL;
	ARlrArmSlowPullJogDcc					: ARRAY [1..iArmSlowPullQty] OF LREAL;

(* xxxxxxxxxxxxxxxxxxxxxxxxxxxxxxxxxxxx Homing Variable xxxxxxxxxxxxxxxxxxxxxxxxxxxxxxxxxxxx*)
(*============================================================================*)

	ARrVertHomeDccDelayTimeSec				: ARRAY [0..iArmQty] OF REAL;
	ARrHorzHomeDccDelayTimeSec				: ARRAY [0..iArmQty] OF REAL;

	ARrArmVertHome1stPercent				: ARRAY [0..iArmQty] OF REAL;
	ARrArmVertHome1stPercentAcc				: ARRAY [0..iArmQty] OF REAL;
	ARrArmVertHome1stPercentDcc				: ARRAY [0..iArmQty] OF REAL;

	ARrArmVertHome2ndPercent				: ARRAY [0..iArmQty] OF REAL;
	ARrArmVertHome2ndPercentAcc				: ARRAY [0..iArmQty] OF REAL;
	ARrArmVertHome2ndPercentDcc				: ARRAY [0..iArmQty] OF REAL;

	ARrArmHorzHome1stPercent				: ARRAY [0..iArmQty] OF REAL;
	ARrArmHorzHome1stPercentAcc				: ARRAY [0..iArmQty] OF REAL;
	ARrArmHorzHome1stPercentDcc				: ARRAY [0..iArmQty] OF REAL;

	ARrArmHorzHome2ndPercent				: ARRAY [0..iArmQty] OF REAL;
	ARrArmHorzHome2ndPercentAcc				: ARRAY [0..iArmQty] OF REAL;
	ARrArmHorzHome2ndPercentDcc				: ARRAY [0..iArmQty] OF REAL;

(* xxxxxxxxxxxxxxxxxxxxxxxxxxxxxxxxx ArmHorzZoneConfirm xxxxxxxxxxxxxxxxxxxxxxxxxxxxxxxxx*)
(*============================================================================*)

	ARlrArmHorzStartPoint 					: ARRAY [0..iArmQty] OF LREAL;
	ARlrArmHorzEndPoint 					: ARRAY [0..iArmQty] OF LREAL;

	ARiArmCurrentHorzZoneNo 				: ARRAY [0..iArmQty] OF INT;
	ARbArmInvalidListingErr					: ARRAY [0..iArmQty] OF BOOL;

	ARlrLdHorzCentrePoint 					: ARRAY [0..iLdStnQty] OF LREAL;
	ARlrStnHorzCentrePoint 					: ARRAY [0..iStnQty] OF LREAL;
	ARlrUldHorzCentrePoint 					: ARRAY [0..iUldStnQty] OF LREAL;

	ARbLdHorzZoneConfirm 					: ARRAY [0..iLdStnQty] OF BOOL;
	ARbArm1HorzStnZoneConfirm 				: ARRAY [1..iStnQty] OF BOOL;
	ARbUldHorzZoneConfirm 					: ARRAY [0..iUldStnQty] OF BOOL;

	ARiArm1HorzListing 						: ARRAY [1..50] OF INT;


(* xxxxxxxxxxxxxxxxxxxxxxxxxxxxxxx Pos Num xxxxxxxxxxxxxxxxxxxxxxxxxxxxxxx*)
(*=========================Pos num============================*)

	ARrVertPos_In_TargetSpdHz				: ARRAY [0..iArmQty] OF REAL;
	ARrVertPos_In_2ndSpdHz					: ARRAY [0..iArmQty] OF REAL;

	ARrHorzPos_In_TargetSpdHz				: ARRAY [0..iArmQty] OF REAL;
	ARrHorzPos_In_2ndSpdHz					: ARRAY [0..iArmQty] OF REAL;

(*=========================Arm Servo Ctrl============================*)

	ARlrVertPos_In_HighSpeed 				: ARRAY [1..iArmQty] OF LREAL;
	ARlrVertPos_In_Acc						: ARRAY [1..iArmQty] OF LREAL;
	ARlrVertPos_In_Dcc						: ARRAY [1..iArmQty] OF LREAL;

	ARlrHorzPos_In_HighSpeed 				: ARRAY [1..iArmQty] OF LREAL;
	ARlrHorzPos_In_Acc						: ARRAY [1..iArmQty] OF LREAL;
	ARlrHorzPos_In_Dcc						: ARRAY [1..iArmQty] OF LREAL;

(* xxxxxxxxxxxxxxxxxxxxxxxxxxxxx Arm Move Variable xxxxxxxxxxxxxxxxxxxxxxxxxxxxxxxxxxxxxx*)
(*============================================================================*)

	DS_ArmLifterPosition					: DS_ArmPnPInOut;

	DSArm1VertConfig						: DS_Servo ;
	DSArm1HorzConfig						: DS_Servo ;

	DSArm2VertConfig						: DS_Servo ;
	DSArm2HorzConfig						: DS_Servo ;

(* xxxxxxxxxxxxxxxxxxxxxxxxxxxxx Generate Arm Pick Transfer Bit xxxxxxxxxxxxxxxxxxxxxxxxxxxxx*)
(*============================================================================*)

	bArmPickLd 								: BOOL;
	bArmPickUld 							: BOOL;
	ARbArmPickStn 							: ARRAY [1..iStnQty] OF BOOL;
	bArmTransferLd 							: BOOL;
	bArmTransferUld 						: BOOL;
	ARbArmTransferStn 						: ARRAY [1..iStnQty] OF BOOL;

(* xxxxxxxxxxxxxxxxxxxxxxxxxxxxx HMI Simulate Arm Movement xxxxxxxxxxxxxxxxxxxxxxxxxxxxx*)
(*============================================================================*)

	lrAngleRatio 							: LREAL;
	bHMIArmSimulateEN 						: BOOL;
	iInterval_ms 							: INT;
	lrMaxSimulateNo 						: LREAL;

	lrSimulateHorzXPos						: LREAL;
	lrSimulateVertYPos						: LREAL;

(* xxxxxxxxxxxxxxxxxxxxxxxxxxxxxxxxxx PnP control variable xxxxxxxxxxxxxxxxxxxxxxxxxxxxxxxxxx*)
(*============================================================================*)

(*Input*)

	ARbPnPStart								: ARRAY [0..iArmQty] OF BOOL;
	ARiPickStnNo							: ARRAY [0..iArmQty] OF INT;
	ARiTransferStnNo						: ARRAY [0..iArmQty] OF INT;
	ARbArmReset								: ARRAY [0..iArmQty] OF BOOL;
	ARbDownPickCondition					: ARRAY [0..iArmQty] OF BOOL;
	ARbDownTransferCondition				: ARRAY [0..iArmQty] OF BOOL;
	ARbPickMidDownStnEn						: ARRAY [0..iStnQty] OF BOOL;
	ARbTransferMidDownStnEn					: ARRAY [0..iStnQty] OF BOOL;
	ARiStationDippingTime					: ARRAY [0..iStnQty] OF INT;
	ARiStepDelayTime						: ARRAY [0..iArmQty] OF INT;

(*Output*)

	ARbArmPnPCompleted						: ARRAY [0..iArmQty] OF BOOL;
	ARbPnPbusy								: ARRAY [0..iArmQty] OF BOOL;

	bMoveTop								: BOOL;
	ARbMoveLdDown							: ARRAY [0..iLdStnQty] OF BOOL;
	ARbMoveUldDown							: ARRAY [0..iUldStnQty] OF BOOL;
	ARbMoveStnMidDown 						: ARRAY [0..iStnQty] OF BOOL;
	ARbMoveStnDown							: ARRAY [0..iStnQty] OF BOOL;

	ARbMoveLdHook							: ARRAY [0..iLdStnQty] OF BOOL;
	ARbMoveLdUnhook							: ARRAY [0..iLdStnQty] OF BOOL;
	ARbMoveStnHook							: ARRAY [0..iStnQty] OF BOOL;
	ARbMoveStnUnhook						: ARRAY [0..iStnQty] OF BOOL;
	ARbMoveUldHook							: ARRAY [0..iUldStnQty] OF BOOL;
	ARbMoveUldUnhook						: ARRAY [0..iUldStnQty] OF BOOL;

	iArm1PnpStep							: INT;
	tStepDelayTimeEV						: TIME;
	iStationDrippingTimeEV					: INT;
	sStatusMessage							: STRING(50);


END_STRUCT
END_TYPE

// ---- DUTs/DS Twincat 3/DS_XML_Persistent_Barcode.TcDUT
TYPE DS_XML_Persistent_Barcode :
STRUCT
	
	ARsProgramDescrip							: ARRAY [0..iProductRecipeArrayQty] OF STRING;
	ARsBarcodeOutput							: ARRAY [0..iProductRecipeArrayQty] OF STRING;
	ARsBarcodeBatch								: ARRAY [0..iProductRecipeArrayQty] OF STRING;
	ARsBarcodeJob								: ARRAY [0..iProductRecipeArrayQty] OF STRING;

	ilengthElimater								: INT :=1;
	bBarcodeBypass								: BOOL;
	bBarcodeEnable 								: BOOL;
	
//V3 Barcode Scanner
	
	DsAr1sG_BarcodeRegistration 				: ARRAY [1..iBarcodeRegQty] 								OF 	DSV3_BarcodeRegistration;
	bBarcodeReceiveStringRst					: BOOL;
	sBarcodeScannerReceivedCmdForReg			: STRING;	
	fbG_BarcodeScanner							: fb_V3BarcodeMasterCtrl;
	
(* xxxxxxxxxxxxxxxxxxxxxxxxxxx fb_V1BarcodeRegistration_UTAC Variable xxxxxxxxxxxxxxxxxxxxxxxxxxx*)
(*=========================================================================*)

	arProgramDescrip1							: ARRAY [0..50] 											OF STRING;

(* xxxxxxxxxxxxxxxxxxxxxxxxxxx fb_V3StringEliminator Variable xxxxxxxxxxxxxxxxxxxxxxxxxxx*)
(*=========================================================================*)

	fbG_V3StringEliminator 						: fb_V3StringEliminator;

	bStringEliminatorEn							: BOOL;
	iCharEliminateQty 							: INT;
	iCharNeededQty								: INT;

(* xxxxxxxxxxxxxxxxxxxxxxxxxxx fb_V3BarcodeRegistration Variable xxxxxxxxxxxxxxxxxxxxxxxxxxx*)
(*==============================================================================*)

	fbG_V1BarcodeRegistration 					: fb_V1BarcodeRegistration_UTAC;

(* xxxxxxxxxxxxxxxxxxxxxxxxxxx fb_V3BarcodeTracer Variable xxxxxxxxxxxxxxxxxxxxxxxxxxx*)
(*==============================================================================*)

	fbG_V3BarcodeTracer 						: fb_V3BarcodeTracer;

	bTracerEn									: BOOL;


(* xxxxxxxxxxxxxxxxxxxxxxxxxxx fb_V3BarcodeRegSectionDisplayController Variable xxxxxxxxxxxxxxxxxxxxxxxxxxx*)
(*=============================================================================================*)

	fbG_V3BarcodeRegSectionDisplayController 	: fb_V3BarcodeRegSectionDisplayController;

	DsAr1sG_BarcodeRegSectionDisplayHMI 		: ARRAY [0..iBarcodeRegSecDisplayQty] 						OF 	DSV3_BarcodeRegistration;
	iAr1sG_BarcodeRegNoSectionDisplayHMI 		: ARRAY [0..iBarcodeRegSecDisplayQty] 						OF 	INT;

	bBarcodeRegEn 								: BOOL;



END_STRUCT
END_TYPE

// ---- DUTs/DS Twincat 3/DS_XML_Persistent_Deactivate.TcDUT
TYPE DS_XML_Persistent_Deactivate :
STRUCT
	
         
                                          
	
	DE10100  : BOOL;   // STN 01 ULTRASONIC GENERATOR ON/OFF (-10U1)     
	DE10101  : BOOL;   // STN 02 ULTRASONIC GENERATOR ON/OFF (-11U1)     
	DE10102  : BOOL;   // STN 04 ULTRASONIC GENERATOR ON/OFF (-12U1)     
	DE10103  : BOOL;   // STN 05 ULTRASONIC GENERATOR ON/OFF (-13U1)     
	DE10104  : BOOL;   // STN 07 ULTRASONIC GENERATOR ON/OFF (-14U1)     
	DE10105  : BOOL;   // STN 08 ULTRASONIC GENERATOR ON/OFF (-15U1)     
	DE10106  : BOOL;   // STN 07 DI WATER RETURN TANK PUMP ON/OFF (-81K1)
	DE10107  : BOOL;   // STN 01 PROCESS TANK PUMP ON/OFF (-73K1)        
	DE10108  : BOOL;   // STN 02 PROCESS TANK PUMP ON/OFF (-74K1)        
	DE10109  : BOOL;   // STN 03 PROCESS TANK PUMP ON/OFF (-75K1)        
	DE10110  : BOOL;   // STN 04 PROCESS TANK PUMP ON/OFF (-76K1)        
	DE10111  : BOOL;   // STN 05 PROCESS TANK PUMP ON/OFF (-77K1)        
	DE10112  : BOOL;   // STN 06 PROCESS TANK PUMP ON/OFF (-78K1)        
	DE10113  : BOOL;   // STN 07 PROCESS TANK PUMP ON/OFF (-79K1)        
	DE10114  : BOOL;   // STN 08 PROCESS TANK PUMP ON/OFF (-80K1)        
	DE10115  : BOOL;   // STN 01 PROCESS TANK HEATER ON/OFF (-130K1)     
	
	DE10200  : BOOL;   // STN 02 PROCESS TANK HEATER ON/OFF (-131K1) 
	DE10201  : BOOL;   // STN 03 PROCESS TANK HEATER ON/OFF (-132K1) 
	DE10202  : BOOL;   // STN 04 PROCESS TANK HEATER ON/OFF (-133K1) 
	DE10203  : BOOL;   // STN 05 PROCESS TANK HEATER ON/OFF (-134K1) 
	DE10204  : BOOL;   // STN 06 PROCESS TANK HEATER ON/OFF (-135K1) 
	DE10205  : BOOL;   // STN 07 PROCESS TANK HEATER ON/OFF (-136K1) 
	DE10206  : BOOL;   // STN 08 PROCESS TANK HEATER ON/OFF (-137K1) 
	DE10207  : BOOL;   // STN 10 PROCESS TANK HEATER ON/OFF (-138K1) 
	DE10208  : BOOL;   // STN 09 - STN 10 FFU UNIT ON/OFF (-163K1)   
	DE10209  : BOOL;   // UNLOADING FFU UNIT ON/OFF (-164K1)         
	DE10210  : BOOL;   // UNLOADING CONVEYOR FFU UNIT ON/OFF (-165K1)
	DE10211  : BOOL;   // STN 09 PROCESS TANK PUMP ON/OFF (-82K1)    

	DE10300  : BOOL;   // STN 01 - 08 AGITATION MOTOR ON/OFF (-160K1)
//	DE10301  : BOOL;   // LOADING CONVEYOR 01 ON/OFF (-170K1)        
//	DE10302  : BOOL;   // LOADING CONVEYOR 02 ON/OFF (-171K1)        
//	DE10303  : BOOL;   // LOADING CONVEYOR 03 ON/OFF (-172K1)        
//	DE10304  : BOOL;   // LOADING CONVEYOR 04 ON/OFF (-173K1)        
//	DE10305  : BOOL;   // UNLOADING CONVEYOR 01 ON/OFF (-174K1)      
//	DE10306  : BOOL;   // UNLOADING CONVEYOR 02 ON/OFF (-175K1)      
//	DE10307  : BOOL;   // UNLOADING CONVEYOR 03 ON/OFF (-176K1)      
//	DE10308  : BOOL;   // UNLOADING CONVEYOR 04 ON/OFF (-177K1)                  
	                    
	
	DE11100  : BOOL;   // STN 03 MEGASONIC GENERATOR 01 ON/OFF (-16U1)
	DE11101  : BOOL;   // STN 03 MEGASONIC GENERATOR 02 ON/OFF (-17U1)
	DE11102  : BOOL;   // STN 01 DOSING PUMP ON/OFF (-70K1)           
	DE11103  : BOOL;   // STN 03 DOSING PUMP ON/OFF (-71K1)           
                      
	
	DE12000  : BOOL;   // STN 05 DOSING PUMP ON/OFF (-72K1)           
	DE12001  : BOOL;   // STN 06 MEGASONIC GENERATOR 01 ON/OFF (-18U1)
	DE12002  : BOOL;   // STN 06 MEGASONIC GENERATOR 02 ON/OFF (-19U1)
	DE12003  : BOOL;   // STN 06 MEGASONIC GENERATOR 03 ON/OFF (-20U1)
                         

                                  


END_STRUCT
END_TYPE

// ---- DUTs/DS Twincat 3/DS_XML_Persistent_Digital.TcDUT
TYPE DS_XML_Persistent_Digital :
STRUCT
	
(* xxxxxxxxxxxxxxxxxxxxxxxxxxxxxxxx DEACTIVATED/BYPASS xxxxxxxxxxxxxxxxxxxxxxxxxxxxxxxx*)
(*========================================================================*)


	ARbArmMissHookByPass1				: ARRAY [1..iArmQty] OF BOOL;
	ARbArmMissHookByPass2				: ARRAY [1..iArmQty] OF BOOL;
	ARbConductivityBypass				: ARRAY [1..iStnQty] OF BOOL;
	ARbFilterPressureBypass				: ARRAY [1..iStnQty] OF BOOL;
	bSafetyDoorSensorBypass				: BOOL;
	ARlrArmDetectZoneRange				: ARRAY [1..iStnQty] OF LREAL;
	ARlrArmStnDetectZoneRange			: ARRAY [1..iArmQty,1..iStnQty] OF LREAL;
	ARiArmDeactDetectZoneRange			: ARRAY [1..iArmQty] OF INT;
	ARbArmMisshook1Alarm				: ARRAY [1..iArmQty] OF BOOL;
	ARbArmMisshook2Alarm				: ARRAY [1..iArmQty] OF BOOL;
	ARbStationFunctionBypass			: ARRAY [1..iStnQty] OF BOOL;
	bStnLiftoutMechanismBypass			: BOOL;
	bBuzzerDisable						: BOOL;
	bUnloadingBuzzerDisable				: BOOL;


END_STRUCT
END_TYPE

// ---- DUTs/DS Twincat 3/DS_XML_Persistent_Memory.TcDUT
TYPE DS_XML_Persistent_Memory :
STRUCT
(* xxxxxxxxxxxsxxxxxx BasketMemory - Basket Cfm/ Trf Internal Used xxxxxxxxsxxxxxxxxx*)
(*========================================================================*)

	fbLdBasketMemory					: ARRAY [0..iCvLdQty] OF fbV2_SingleArmBasketMemoryV2;
	fbA1StationBasketMemory				: ARRAY [0..iStnQty] OF fbV2_SingleArmBasketMemoryV2;
	fbA2StationBasketMemory				: ARRAY [0..iStnQty] OF fbV2_SingleArmBasketMemoryV2;
	fbUldBasketMemory					: ARRAY [0..iCvUldQty] OF fbV2_SingleArmBasketMemoryV2;

(* xxxxxxxxxxxxxxxxxxxxxxxxxxxx  BasketInfo - Internal Used xxxxxxxxxxxxxxxxxxxxxxxxxxxx*)
(*========================================================================*)

	DSLdBasketInfoConfirm 				: ARRAY [0..iLdStnQty] OF DSV2_BasketInfo;
	DSLdBasketInfoTransfer 				: ARRAY [0..iLdStnQty] OF DSV2_BasketInfo;

	DSUldBasketInfoConfirm 				: ARRAY [0..iUldStnQty] OF DSV2_BasketInfo;
	DSUldBasketInfoTransfer 			: ARRAY [0..iUldStnQty] OF DSV2_BasketInfo;

	DSStnBasketInfo						: ARRAY [0..iStnQty] OF DSV2_BasketInfo;
	DSArmBasketInfo 					: ARRAY [0..iArmQty] OF DSV2_BasketInfo;

(* xxxxxxxxxxxxxxxxxxxxx  BasketInfo - Loading / Unloading Conveyor Used xxxxxxxxxxxxxxxxxxxxx *)
(*================================================================================*)

	AR2sDSCv_LdConfirmBasketInfo 		: ARRAY [1..iLdStnQty, 1..iCvLdQty] OF DSV2_BasketInfo;
	AR2sDSCv_LdTransferBasketInfo 		: ARRAY [1..iLdStnQty, 1..iCvLdQty] OF DSV2_BasketInfo;

	AR2sDSCv_UldConfirmBasketInfo 		: ARRAY [1..iUldStnQty, 1..iCvUldQty] OF DSV2_BasketInfo;
	AR2sDSCv_UldTransferBasketInfo 		: ARRAY [1..iUldStnQty, 1..iCvUldQty] OF DSV2_BasketInfo;

(* xxxxxxxxxxxxxxxxxxxxx  Station Memory and InputOutput Variable - Internal Used xxxxxxxxxxxxxxxxxxxxx*)
(*=====================================================================================*)

	LdDSStationSSERStore				: DSV2_fbStationSequenceRecipeStore;
	LdDSStationSSURStore 				: DS_fbStationSubRecipeStore;

	LdDSStationSSERCall					: DSV2_fbStationSequenceRecipeCall;
	LdDSStationSSURCall 				: DS_fbStationSubRecipeCall;

	ARDsStnSeqProInput 					: ARRAY [0..iStnQty] OF DS_StnSeqProInput;
	ARDSStnSeqProOutput 				: ARRAY [0..iStnQty] OF DS_StnSeqProOutput;

	AR10DSStationSSERStore				: ARRAY [0..iStnQty] OF DSV2_fbStationSequenceRecipeStore;
	AR10DSStationSSERCall				: ARRAY [0..iStnQty] OF DSV2_fbStationSequenceRecipeCall;

	AR10DSStationSSURStore 				: ARRAY [0..iStnQty] OF DS_fbStationSubRecipeStore;
	AR10DSStationSSURCall 				: ARRAY [0..iStnQty] OF DS_fbStationSubRecipeCall;

(* xxxxxxxxxxxxxxxxxxxxxxxxxxxxx  Station Process Variable - Internal Used xxxxxxxxxxxxxxxxxxxxxxxxxxxxx*)
(*=====================================================================================*)

	fbMainStationProcess_Stn			: ARRAY [1..iStnQty] OF fbV2_MainStationProcess;
	ARDsStnSeqProcessCtrl 				: ARRAY [0..iStnQty] OF DS_fbStnSeqProcessCtrl;
	ARbProductRecipeCallEn 				: ARRAY [0..iStnQty] OF BOOL;
	ARiProductRecipeNoCall 				: ARRAY [0..iStnQty] OF INT;
	ARiProductRecipeStepCall 			: ARRAY [0..iStnQty] OF INT;
	DSfbGnrProductRecipeMemoryOut 		: DSV2_fbGnrProductRecipeMemoryOut;
	ARiStnNoToCalledArm					: ARRAY [0..iArmQty] OF INT;
	ARDSGnrFeedArmPnpParameter			: ARRAY [0..iArmQty] OF DSV2_Gnr_CalledArmPnpParameter;
	ARbArmReady							: ARRAY [1..iArmQty] OF BOOL;(* Universal*) (* Input  - From ArmPnpFB, This signal is used to confirm if the arm is ready and idling*)
	ARbStationProcessCompletedFlag		: ARRAY [0..iStnQty] OF BOOL;

(*xxxxxxxxxxxxxxxxxxxxxxxxxxx fbGnrProductRecipeMemory - Internal Used xxxxxxxxxxxxxxxxxxxxxxxxxxx*)
(*=====================================================================================*)

(*Input/Output*)
	ARiCurrentHorzStnNo					: ARRAY [1..iArmQty] OF INT;
	ARi1StepPatternNo					: ARRAY [1..iArmQty] OF INT;
	ARDs1StepUpDownMovement				: ARRAY [1..iArmQty] OF DSA1_UpDownMovement;
	ARi4StepPatternNo					: ARRAY [1..iArmQty] OF INT;
	ARDs4StepUpDownMovement				: ARRAY [1..iArmQty] OF DSA1_UpDownMovement;

(* xxxxxxxxxxxxxxxxxxxxxxxxxxx  Station ZoneHeight Variable - External Used xxxxxxxxxxxxxxxxxxxxxxxxxxx*)
(*=====================================================================================*)

	ARDSLdZoneHeight 					: ARRAY [0..iLdStnQty] OF DSA32_StationZoneHeight;
	ARDSStationZoneHeight 				: ARRAY [0..iStnQty] OF DSA32_StationZoneHeight;
	ARDSUldZoneHeight 					: ARRAY [0..iUldStnQty] OF DSA32_StationZoneHeight;

(* xxxxxxxxxxxxxxxxxxxxxxxxxxx  Station ZoneHeight Variable - Internal Used xxxxxxxxxxxxxxxxxxxxxxxxxxx*)
(*=====================================================================================*)

	ARDSLdZonePosOut					: ARRAY [0..iLdStnQty] OF DSA32_StationZonePosOut; (*From fbGnrProductRecipeMemory Output*)
	ARDSStationZonePosOut 				: ARRAY [0..iStnQty] OF DSA32_StationZonePosOut; (*From fbGnrProductRecipeMemory Output*)
	ARDSUldZonePosOut 					: ARRAY [0..iUldStnQty] OF DSA32_StationZonePosOut;(*From fbGnrProductRecipeMemory Output*)

(* xxxxxxxxxxxxxxxxxxxxxxxxxxxxx  MaxMin Time Used  xxxxxxxxxxxxxxxxxxxxxxxxxxxxx*)
(*====================================================================*)

	ARDsSSERSourceMinMaxTime_Uni		: ARRAY [1..iStnQty] OF DSV2_SSERSourceMinMaxTime;
	ARDsStnMinMaxEffTimeDisplay			: ARRAY [0..iStnQty] OF DSV2_StnMinMaxEffTIme;
	DSV2MTBMinMaxEffTime 				: DSV2_MinMaxEffTime;


END_STRUCT
END_TYPE

// ---- DUTs/DS Twincat 3/DS_XML_Persistent_Process.TcDUT
TYPE DS_XML_Persistent_Process :
STRUCT
	(* xxxxxxxxxxxxxxxxxxxxxxx DosingPumpControl Process Variable xxxxxxxxxxxxxxxxxxxxxxx*)
(*========================================================================*)

	ARDSProminentDosingHMI 									: ARRAY [1..iStnQty] OF DS_ProminentDosingHMI;
	ARfbProminentDosingCtrl									: ARRAY [1..iStnQty] OF fbProminentDosingCtrl;

	ARiStnPulseOnTime_ms									: ARRAY [1..iStnQty] OF INT;
	ARiStnPulseOffTime_ms 									: ARRAY [1..iStnQty] OF INT;
	ARiStnPumpFeedbackPulseInputFilter_ms 					: ARRAY [1..iStnQty] OF INT;
	ARiStnPumpHealthCheckPulseSV 							: ARRAY [1..iStnQty] OF INT;

(* xxxxxxxxxxxxxxxxxxxxxxxxxxxxx Conveyor Motor Control xxxxxxxxxxxxxxxxxxxxxxxxxxxxx*)
(*========================================================================*)

	ARrLdIndexPBDelayTimeSV_Sec 							: ARRAY [0..iLdStnQty] OF REAL;
	ARrLdRapidPBDelayTimeSV_Sec 							: ARRAY [0..iLdStnQty] OF REAL;
	ARrLdIndexConfirmDelayTimeSV_Sec 						: ARRAY [0..iLdStnQty] OF REAL;
	ARrLdEndZoneDelayTimeSV_Sec 							: ARRAY [0..iLdStnQty] OF REAL;

	ARrUldIndexPBDelayTimeSV_Sec 							: ARRAY [0..iUldStnQty] OF REAL;
	ARrUldRapidPBDelayTimeSV_Sec 							: ARRAY [0..iUldStnQty] OF REAL;
	ARrUldIndexConfirmDelayTimeSV_Sec 						: ARRAY [0..iUldStnQty] OF REAL;
	ARrUldEndZoneDelayTimeSV_Sec 							: ARRAY [0..iUldStnQty] OF REAL;

	diUnloadingTimer										: DINT;
	iUldBasketDelayPushTimerSV_sec							: INT;
	iUldBasketDelayPushTimeCountDown						: INT;
	diLdReturnConvMotorDelayOffTimer						: DINT;
	diUldReturnConvMotorDelayOffTimer						: DINT;

	rLdConveyorPos1ConfirmDelayTimeSV_Sec 					: REAL;
	rLdConveyorPos2ConfirmDelayTimeSV_Sec 					: REAL;
	rLdConveyorPos3ConfirmDelayTimeSV_Sec 					: REAL;
	rLdConveyorPos4ConfirmDelayTimeSV_Sec 					: REAL;

	rLdConveyorPos1ConfirmDelayOnTimeSV_Sec 				: REAL;
	rLdConveyorPos2ConfirmDelayOnTimeSV_Sec 				: REAL;
	rLdConveyorPos3ConfirmDelayOnTimeSV_Sec 				: REAL;
	rLdConveyorPos4ConfirmDelayOnTimeSV_Sec 				: REAL;
	
	rUldConveyorPos1ConfirmDelayTimeSV_Sec 					: REAL;
	rUldConveyorPos2ConfirmDelayTimeSV_Sec 					: REAL;
	rUldConveyorPos3ConfirmDelayTimeSV_Sec 					: REAL;
	rUldConveyorPos4ConfirmDelayTimeSV_Sec 					: REAL;

	rUldConveyorPos1ConfirmDelayOnTimeSV_Sec 				: REAL;
	rUldConveyorPos2ConfirmDelayOnTimeSV_Sec 				: REAL;
	rUldConveyorPos3ConfirmDelayOnTimeSV_Sec 				: REAL;
	rUldConveyorPos4ConfirmDelayOnTimeSV_Sec 				: REAL;
	
(* xxxxxxxxxxxxxxxxxxxxxxxxxxx General Process Variable xxxxxxxxxxxxxxxxxxxxxxxxxxx*)
(*======================================================================*)

	ARiStnToleranceTimeSV									: ARRAY [0..iStnQty] OF INT;
	ARiArmToleranceTimeSV									: ARRAY [0..iArmQty] OF INT;

	ARbRecipeSelectedFlag									: ARRAY [1..iProductRecipeArrayQty] OF BOOL;

    ARbOptionSelectedAutoTopupFlag							: ARRAY [1..iProductRecipeArrayQty] OF BOOL;
    ARbOptionSelectedRecipeFlag								: ARRAY [1..iProductRecipeArrayQty] OF BOOL;

(* xxxxxxxxxxxxxxxxxxxxxxxxxxx Arm related in Process xxxxxxxxxxxxxxxxxxxxxxxxxxx*)
(*======================================================================*)

	tAllStnArmTake											: INT;
	ARiStnDippingTimeSV										: ARRAY [1..iStnQty] OF INT;
	iFFUDelayOffTimerSV_min									: INT;
	iStnAgitation1DelayOffTimerSV_min						: INT;
	iStnAgitation2DelayOffTimerSV_min						: INT;

(* xxxxxxxxxxxxxxxxxxxxxxxxxxxxx Valve related in Process  xxxxxxxxxxxxxxxxxxxxxxxxxxxxx*)

	iAllTankLowLevelDelayTimeSV 							: INT;
	ARiStnTopUpDelayOffTimeSV								: ARRAY [1..iStnQty] OF INT;
	ARiStnSubTankTopUpDelayOffTimeSV						: ARRAY [1..iStnQty] OF INT;

	ARiStnTopUpMaxTimeCutOffSV								: ARRAY [1..iStnQty] OF INT;

	iVacuumDrainSV											: INT;

	bBasketPushBasedTimer									: BOOL;

	ARbIncomingDIValveBasedDetergent						: ARRAY [1..iStnQty] OF BOOL;

	iCylinderBasketBackDelayTimeSV							: INT;
	iCylinderBasketFrontDelayTimeSV							: INT;

	iStn3PumpHzSV											: INT;


END_STRUCT
END_TYPE

// ---- DUTs/DS Twincat 3/DS_XML_Persistent_SevenDay.TcDUT
TYPE DS_XML_Persistent_SevenDay :
STRUCT
	TodayDay 				: STRING;

	ArbDayOnEn_IN			: ARRAY [1..7] OF BOOL;
	ArbDayOffEn_IN			: ARRAY [1..7] OF BOOL;

	ArwDayOnHour_IN			: ARRAY [1..7] OF WORD;
	ArwDayOnMinute_IN		: ARRAY [1..7] OF WORD;

	ArwDayOffHour_IN		: ARRAY [1..7] OF WORD;
	ArwDayOffMinute_IN		: ARRAY [1..7] OF WORD;

	ArbDaySysOn_OUT			: ARRAY [1..7] OF BOOL;
	ArbDaySysOff_OUT		: ARRAY [1..7] OF BOOL;
END_STRUCT
END_TYPE

// ---- DUTs/DS Twincat 3/DS_XML_Persistent_TimeOptimize.TcDUT
TYPE DS_XML_Persistent_TimeOptimize :
STRUCT
	
	bTimeOptimizeDisable								: BOOL;

	ARiCalledTotalProcessTimeStn1						: ARRAY[1..5] OF INT;
	ARiCalledTotalProcessTimeStn2						: ARRAY[1..5] OF INT;
	ARiCalledTotalProcessTimeStn3						: ARRAY[1..5] OF INT;
	ARiCalledTotalProcessTimeStn4						: ARRAY[1..5] OF INT;
	ARiCalledTotalProcessTimeStn5						: ARRAY[1..5] OF INT;
	ARiCalledTotalProcessTimeStn6						: ARRAY[1..5] OF INT;
	ARiCalledTotalProcessTimeStn7						: ARRAY[1..5] OF INT;
	ARiCalledTotalProcessTimeStn8						: ARRAY[1..5] OF INT;
	ARiCalledTotalProcessTimeStn9						: ARRAY[1..5] OF INT;
	ARiCalledTotalProcessTimeStn10						: ARRAY[1..5] OF INT;

(*[][][][][][][][][][][][][][][][][][][][]---fbMasterTimeBlockG2---[][][][][][][][][][][][][][][][][][][][]*)
(*
	fbV2MasterTimeBlockG2_Auto							: fbV2_MasterTimeBlockG2;
*)
(*Input*)
	bMTBStartEN 										: BOOL;
	bMTBScanEN											: BOOL;                         (*bScanOnFlag*)
	bMTBWriteEN 										: BOOL;
	bMTBResetEN 										: BOOL;

(*Output*)
	bMTBScanCompletedFlag								: BOOL;
	bMTBWriteDoneFlag 									: BOOL;
	bMTBResetDoneFlag 									: BOOL;
	bMTBWriteArmDataError 								: BOOL;
	bMTBWriteStnDataError								: BOOL;
	bMTBWriteUldDataError								: BOOL;
	bMTBNoAvailableSlotError 							: BOOL;
	bMTBArmIDAndStnIDAndUldIDNotFound				 	: BOOL;

	bMTBWriteDisable									: BOOL;
	bMTBWriteRetry										: BOOL;
	bMTBWriteExecuteError								: BOOL;

	iMTBNextTransferScanCounter							: INT;
	iMTBNextNotAvailableScanCounter						: INT;
	iMTBNextTransferTime								: INT;
	iMTBNextNotAvailableTime							: INT;

(*[][][][][][][][][][][][][][][][][][][][]---fbTimeBlockSimulatorG2---[][][][][][][][][][][][][][][][][][][][]*)

	fbV2TimeBlockSimulatorG2_Main						: fbV2_TimeBlockSimulatorG2;

(*Input*)
	bSimulateTSEN										: BOOL;

(*Output*)
	bSimulateCompletedFlag								: BOOL;
	iSimulatePercentage									: INT;
	bSimNoSpaceForArmDataToFill							: BOOL;
	bSimNoSpaceForStnDataToFill							: BOOL;
	bSimArmIDAndStnIDNotFound							: BOOL;

	iSimulatedBasketQty									: INT;
	iSimMasterTotalTime									: INT;
	iSimAvarageTimeSec									: INT;

	rSimBasketQtyPerHour								: REAL;

(*[][][][][][][][][][][][][][][][][][][][]---fbFBPTimeTrackerG2---[][][][][][][][][][][][][][][][][][][][]*)

	DSTimeTrackerInput									: DSV2_TimeTrackerInput;

(*Input*)
	bTrackerStartEN										: BOOL;

	iCallRecipeTimeBlock_ProductRecipeNo 				: INT;

	iSimulatorProductRecipeNo							: INT;
	iUserDefineProductRecipeNo							: INT;
	iTrackerProductRecipeNo 							: INT;
	iDisplayUserDefineProductRecipeNo					:INT;

(*Output*)

	bTrackerCompleted 									: BOOL;
	bNoUldStnIDErr										: BOOL;
	bInvalidCallRecipeTimeBlockNo						: BOOL;
	bCallRTB_NoTrackerInfo								: BOOL;
	bCallRTB_CallOK 									: BOOL;
	bCallModeError										: BOOL;


(*[][][][][][][][][][][][][][][][][][][][]---fbMasterTimeBlockG2---[][][][][][][][][][][][][][][][][][][][]*)

(*Input*)
	iMTBScanCompleteDelayOnTime_ms						: INT := 1000;
	iMTBWriteRetryQty									: INT := 3;
	iMTBWriteRetryDelayTimeSec							: INT := 2;

	AR3SiMasterTimeBlockArm_MTB		 					: ARRAY[1..iArmQty, 1..iMasterBlockQty, 1..3] OF INT;
	AR3SiMasterTimeBlockStn_MTB							: ARRAY[1..iStnQty, 1..iMasterBlockQty, 1..3] OF INT;
	AR3SiMasterTimeBlockUld_MTB							: ARRAY[1..iUldStnQty, 1..iMasterBlockQty, 1..3] OF INT;

(*Output*)
	ARbMTBArmProgress									: ARRAY [1..iArmQty] OF BOOL;

(*[][][][][][][][][][][][][][][][][][][][]---fbTimeBlockSimulatorG2---[][][][][][][][][][][][][][][][][][][][]*)

(*Input*)
	AR3SiMasterTimeBlockArm_Simulator 					: ARRAY[1..iArmQty, 1..iMasterBlockQty, 1..9] OF INT;
	AR3SiMasterTimeBlockStn_Simulator					: ARRAY[1..iStnQty, 1..iMasterBlockQty, 1..9] OF INT;

(*Output*)
	ARiSimBasketTimeStamp 								: ARRAY [1..100] OF INT;


(*[][][][][][][][][][][][][][][][][][][][]---fbFBPTimeTrackerG2---[][][][][][][][][][][][][][][][][][][][]*)

	fbV2FBPTimeTrackerG3_Main							: fbV2_FBPTimeTrackerG3;


(*Input*)

	bTrackerReset 										: ARRAY [0..iProductRecipeArrayQty] OF BOOL;

	ARbReset 											: ARRAY [0..iProductRecipeArrayQty] OF BOOL;
	ARbArmSt 											: ARRAY [1..iArmQty] OF BOOL; (*Activated Bit*)
	iCountFilterTime_Sec 								: INT := 2;
	AR2SiBufferRecipeTimeBlock 							: ARRAY[1..iRecipeBlockQty, 1..9] OF INT;

	ARbBusyLinkUpStnEn 									: ARRAY [1..iBusyLinkUpSetQty] OF BOOL;
	AR2siStnBusyLinkUpStn 								: ARRAY [1..iBusyLinkUpSetQty, 1..iBusyLinkUpStnQty] OF INT;


(*Output*)

	AR2SiCalledRecipeTimeBlockNoCallArmTime 			: ARRAY[1..iRecipeBlockQty, 1..9] OF INT;
	AR2SiCalledRecipeTimeBlockWithCallArmTime 			: ARRAY[1..iRecipeBlockQty, 1..9] OF INT;

	ARbProductRecipeTimeBlockAvailable					: ARRAY [0..iProductRecipeArrayQty] OF BOOL;

	AR2SiArmRunningTime									: ARRAY [1..iRecipeBlockQty, 1..iArmQty] OF INT;
	ARiStnRunningTime									: ARRAY [1..iRecipeBlockQty] OF INT;

(*[][][][][][][][][][][][][][][][][][][][]---Multiple FB Used---[][][][][][][][][][][][][][][][][][][][]*)

(*	AR2SiRecipeTimeBlock								: ARRAY [1..iRecipeBlockQty, 1..3] OF INT;
	ARbSkipStation										: ARRAY [1..iStnQty] OF BOOL;

	ARiZoneAddress										: ARRAY [1..iRecipeBlockQty] OF INT;
	ARiZoneArea											: ARRAY [1..iRecipeBlockQty] OF INT;
*)	ARiArmID											: ARRAY [1..iArmQty] OF INT;


(*[][][][][][][][][][][][][][][][][][][][]---fbFBPTimeTrackerG2---[][][][][][][][][][][][][][][][][][][][]*)


(*Input*)
	ARbAlternateStnEn 									: ARRAY [1..iAlternateSetQty] OF BOOL;
	AR2siAlternateStn 									: ARRAY [1..iAlternateSetQty, 1..iAlternateStnQty] OF INT;
END_STRUCT
END_TYPE

// ---- DUTs/DS Twincat 3/Enum/Digital_Input.TcDUT
{attribute 'Tc2GvlVarNames'}
{attribute 'strict'}
{attribute 'to_String'}

TYPE Digital_Input :
(
		eX10000_Stn01_03UltrasonicGeneratorMcb_Trip               			 	   :=1,  
		eX10001_Stn01UltrasonicGeneratorLeftRight_Alarm   	                       :=2,  
		eX10002_Stn01UltrasonicGeneratorBottom_Alarm                               :=3,  
		eX10003_Stn02UltrasonicGeneratorLeftRight_Alarm                            :=4,  
		eX10004_Stn02UltrasonicGeneratorBottom_Alarm                               :=5,  
		eX10005_Stn03UltrasonicGeneratorLeftRight_Alarm                            :=6,  
		eX10006_Stn03UltrasonicGeneratorBottom_Alarm                               :=7,  
		eX10007_Stn04_05UltrasonicGeneratorMcb_Trip                                :=8,  
		eX10008_Stn04UltrasonicGeneratorLeftRight_Alarm                            :=9,  
		eX10009_Stn04UltrasonicGeneratorBottom_Alarm                               :=10, 
		eX10010_Stn05UltrasonicGeneratorBottom_Alarm                               :=11, 
		eX10011_GeneralMainPanelPb_E_Stop                                          :=12, 
		eX10012_OperatorPullString_E_Stop                                          :=13, 
		eX10013_MaintenancePullString_E_Stop                                       :=14, 
		eX10014_GeneralTouchMonitorSocketElcb_Trip                                 :=15, 
		eX10015_Arm01ServoDriveMcb_Trip                                            :=16, 
		                                                                                 
		eX10100_IpcDcOnSignal                                                      :=17, 
		eX10101_PanelVentilationFanMcb_Trip                                        :=18, 
		eX10102_PanelLightingMcb_Trip                                              :=19, 
		eX10103_MachineLighting01Mcb_Trip                                          :=20, 
		eX10104_MachineLighting02Mcb_Trip                                          :=21, 
		eX10105_GeneralTouchMonitorSocketMcb_Trip                                  :=22, 
		eX10106_GeneralPhaseSequenceRelayMcb_Trip                                  :=23, 
		eX10107_GeneralPhaseSequenceRelay_Trip                                     :=24, 
		eX10108_Stn06ProcessTankBlowerMms_Tor_Trip                                 :=25, 
		eX10109_Stn01_06ExhaustBlowerMms_Tor_Trip                                  :=26, 
		eX10110_Stn01_05AgitationMotorMms_Tor_Trip                                 :=27, 
		eX10111_Stn01DosingPumpMcb_Trip                                            :=28, 
		eX10112_Stn02DosingPumpMcb_Trip                                            :=29, 
		eX10113_Stn03DosingPumpMcb_Trip                                            :=30, 
		eX10114_Stn04DosingPumpMcb_Trip                                            :=31, 
		eX10115_Stn01DosingChemicalContainerRelaySignal_Feedback                   :=32, 
		                                                                                 
		eX10200_Stn01ProcessTankPumpMms_Tor_Trip                                   :=33, 
		eX10201_Stn02ProcessTankPumpMms_Tor_Trip                                   :=34, 
		eX10202_Stn03ProcessTankPumpMms_Tor_Trip                                   :=35, 
		eX10203_Stn04ProcessTankPumpMms_Tor_Trip                                   :=36, 
		eX10204_Stn05ProcessTankPumpMms_Tor_Trip                                   :=37, 
		eX10205_Stn01_04ChemicalReturnTankPumpMms_Tor_Trip                         :=38, 
		eX10206_Stn06ProcessTankVacuumPumpMms_Tor_Trip                             :=39, 
		eX10207_Stn01ProcessTankHeaterMcb_Trip                                     :=40, 
		eX10208_Stn02ProcessTankHeaterMcb_Trip                                     :=41, 
		eX10209_Stn03ProcessTankHeaterMcb_Trip                                     :=42, 
		eX10210_Stn04ProcessTankHeaterMcb_Trip                                     :=43, 
		eX10211_Stn06ProcessTankHeaterMcb_Trip                                     :=44, 
		eX10212_LoadingConveyor1Mcb_Trip                                           :=45, 
		eX10213_LoadingConveyor2Mcb_Trip                                           :=46, 
		eX10214_LoadingConveyor3Mcb_Trip                                           :=47, 
		eX10215_Stn02DosingChemicalContainerRelaySignal_Feedback                   :=48, 
		                                                                                 
		eX10300_MainSafetyContactor1_Feedback                                      :=49, 
		eX10301_MainSafetyContactor2_Feedback                                      :=50, 
		eX10302_DoorSafetyContactor1_Feedback                                      :=51, 
		eX10303_DoorSafetyContactor2_Feedback                                      :=52, 
		eX10304_Module01AdditionalPowerSupplyIncomingPowerMcb_Trip                 :=53, 
		eX10305_Module01AdditionalPowerSupplyOutgoingPowerMcb_Trip                 :=54, 
		eX10306_Module02AdditionalPowerSupplyIncomingPowerMcb_Trip                 :=55, 
		eX10307_Module02AdditionalPowerSupplyOutgoingPowerMcb_Trip                 :=56, 
		eX10308_Module03AdditionalPowerSupplyIncomingPowerMcb_Trip                 :=57, 
		eX10309_Module03AdditionalPowerSupplyOutgoingPowerMcb_Trip         		   :=58, 
		eX10310_Arm01AdditionalPowerSupplyIncomingPowerMcb_Trip                    :=59, 
		eX10311_Arm01AdditionalPowerSupplyOutgoingPowerMcb_Trip                    :=60, 
		eX10312_Stn05_06FfuUnitMcb_Trip                                            :=61, 
		eX10313_UnloadingFfuUnitMcb_Trip                                           :=62, 
		eX10314_Reserved                                                           :=63, 
		eX10315_Reserved                                                           :=64, 
		                                                                                 
		eX10400_GeneralAlarmPb_Reset                                               :=65, 
		eX10401_GeneralBuzzerPb_Reset                                              :=66, 
		eX10402_Stn01ProcessTankSensor_MaxOverflow                                 :=67, 
		eX10403_Stn01ProcessTankSensor_MinOverflow                                 :=68, 
		eX10404_Stn01ProcessTankSensor_Min                                         :=69, 
		eX10405_Stn02ProcessTankSensor_MaxOverflow                                 :=70, 
		eX10406_Stn02ProcessTankSensor_MinOverflow                                 :=71, 
		eX10407_Stn02ProcessTankSensor_Min                                         :=72, 
		eX10408_Stn01DosingChemicalContainerSensor_WarningLevel                    :=73, 
		eX10409_Stn01DosingChemicalContainerSensor_MinLevel                        :=74, 
		eX10410_Structure01DripPanSensor_Leak                                      :=75, 
		eX10411_Stn02DosingChemicalContainerSensor_WarningLevel                    :=76, 
		eX10412_Stn02DosingChemicalContainerSensor_MinLevel                        :=77, 
		eX10413_Arm01HorizontalSensor_LoadingOt                                    :=78, 
		eX10414_Arm01HorizontalSensor_Home                                         :=79, 
		eX10415_GeneralSafetyCurtainSensor_Alarm                                   :=80, 
		                                                                                 
		eX11000_Arm01VerticalSensor_TopOt                                          :=81, 
		eX11001_Arm01VerticalSensor_Home                                           :=82, 
		eX11002_Arm01VerticalSensor_BtmOt                                          :=83, 
		eX11003_Arm01VerticalSensor_Crash                                          :=84, 
		eX11004_Arm01SensorA_Misshook                                              :=85, 
		eX11005_Arm01SensorB_Misshook                                              :=86, 
		eX11006_Stn03ProcessTankSensor_MaxOverflow                                 :=87, 
		eX11007_Stn03ProcessTankSensor_MinOverflow                                 :=88, 
		eX11008_Stn03ProcessTankSensor_Min                                         :=89, 
		eX11009_Stn04ProcessTankSensor_MaxOverflow                                 :=90, 
		eX11010_Stn04ProcessTankSensor_Min                                         :=91, 
		eX11011_Structure02DripPanSensor_Leak                                      :=92, 
		eX11012_Stn03DosingChemicalContainerSensor_WarningLevel                    :=93, 
		eX11013_Stn03DosingChemicalContainerSensor_MinLevel                        :=94, 
		eX11014_Stn04DosingChemicalContainerSensor_WarningLevel                    :=95, 
		eX11015_Stn04DosingChemicalContainerSensor_MinLevel                        :=96, 
		                                                                                 
		eX11100_Stn03DosingChemicalContainerRelaySignal_Feedback                   :=97, 
		eX11101_Stn04DosingChemicalContainerRelaySignal_Feedback                   :=98, 
		eX11102_Stn04ProcessTankSensor_MinOverflow                                 :=99, 
		eX11103_Reserved                                                           :=100,
		eX11104_Reserved                                                           :=101,
		eX11105_Reserved                                                           :=102,
		eX11106_Reserved                                                           :=103,
		eX11107_Reserved                                                           :=104,
		eX11108_Reserved                                                           :=105,
		eX11109_Reserved                                                           :=106,
		eX11110_Reserved                                                           :=107,
		eX11111_Reserved                                                           :=108,
		eX11112_Reserved                                                           :=109,
		eX11113_Reserved                                                           :=110,
		eX11114_Reserved                                                           :=111,
		eX11115_Reserved                                                           :=112,
		                                                                                 
		eX12000_Stn05ProcessTankSensor_MaxOverflow                                 :=113,
		eX12001_Stn05ProcessTankSensor_Min                                         :=114,
		eX12002_Stn01_04ChemicalReturnTankSensor_Max                               :=115,
		eX12003_Stn01_04ChemicalReturnTankSensor_Reg                               :=116,
		eX12004_Stn01_04ChemicalReturnTankSensor_Min                               :=117,
		eX12005_Stn05ProcessTankFlowSensor_MinFlow                                 :=118,
		eX12006_Stn06ProcessTankHeaterThermostat_Alarm                             :=119,
		eX12007_Stn06SlidingDoorRs_Open                                            :=120,
		eX12008_Stn06SlidingDoorRs_Close                                           :=121,
		eX12009_Structure03DripPanSensor_Leak                                      :=122,
		eX12010_GeneralIncomingCdaPressureSwitch_MinPressure                       :=123,
		eX12011_UnloadingSensor_BasketDetection                                    :=124,
		eX12012_Arm01HorizontalSensor_UnloadingOt                                  :=125,
		eX12013_Reserved                                                           :=126,
		eX12014_Reserved                                                           :=127,
		eX12015_Reserved                                                           :=128,
		                                                                                 
		eX12100_Stn06SlidingDoorRs01_Clamp                                         :=129,
		eX12101_Stn06SlidingDoorRs01_Unclamp                                       :=130,
		eX12102_Stn06SlidingDoorRs02_Clamp                                         :=131,
		eX12103_Stn06SlidingDoorRs02_Unclamp                                       :=132,
		eX12104_Reserved                                                           :=133,
		eX12105_Reserved                                                           :=134,
		eX12106_Reserved                                                           :=135,
		eX12107_Reserved                                                           :=136,
		eX12108_Reserved                                                           :=137,
		eX12109_Reserved                                                           :=138,
		eX12110_Reserved                                                           :=139,
		eX12111_Reserved                                                           :=140,
		eX12112_Reserved                                                           :=141,
		eX12113_Reserved                                                           :=142,
		eX12114_Reserved                                                           :=143,
		eX12115_Reserved                                                           :=144,
		                                                                                 
		eX13000_LoadingConveyorSensor_Feed                                         :=145,
		eX13001_LoadingConveyorSensor_Index                                        :=146,
		eX13002_LoadingConveyorSensor_Pick                                         :=147,
		eX13003_GeneralLoadingPb_E_Stop                                            :=148,
		eX13004_Reserved                                                           :=149,
		eX13005_Reserved                                                           :=150,
		eX13006_Reserved                                                           :=151,
		eX13007_Reserved                                                           :=152,
		eX13008_Reserved                                                           :=153,
		eX13009_Reserved                                                           :=154,
		eX13010_Reserved                                                           :=155,
		eX13011_Reserved                                                           :=156,
		eX13012_Reserved                                                           :=157,
		eX13013_Reserved                                                           :=158,
		eX13014_Reserved                                                           :=159,
		eX13015_Reserved                                                           :=160
                                                                    	                                                                    
   );
END_TYPE

// ---- DUTs/DS Twincat 3/Enum/Digital_Output.TcDUT
{attribute 'Tc2GvlVarNames'}
{attribute 'strict'}
{attribute 'to_String'}

TYPE Digital_Output :
(
		eY10000_EmergencyStopSafetyRelay_Reset										:=1,  
		eY10001_Stn01_03UltrasonicGeneratorFrequencyChangeBit1                      :=2,  
		eY10002_Stn01_03UltrasonicGeneratorFrequencyChangeBit2                      :=3,  
		eY10003_Stn04_05UltrasonicGeneratorFrequencyChangeBit1                      :=4,  
		eY10004_Stn04_05UltrasonicGeneratorFrequencyChangeBit2                      :=5,  
		eY10005_GeneralAlarmResetInd                                                :=6,  
		eY10006_GeneralBuzzerResetInd                                               :=7,  
		eY10007_GeneralBuzzerTone1                                                  :=8,  
		eY10008_GeneralBuzzerTone2                                                  :=9,  
		eY10009_GeneralTowerLightInd_Red                                            :=10, 
		eY10010_GeneralTowerLightInd_Yellow                                         :=11, 
		eY10011_GeneralTowerLightInd_Green                                          :=12, 
		eY10012_IpcDcOnHoldingRelay                                                 :=13, 
		eY10013_Stn05_06FfuUnitOnOff                                               	:=14, 
		eY10014_UnloadingFfuUnitOnOff                                               :=15, 
		eY10015_Reserved                                                            :=16, 
		                                                                                  
		eY10100_Stn01UltrasonicGeneratorLeftRightOnOff                              :=17,
		eY10101_Stn01UltrasonicGeneratorBottomOnOff                          	    :=18, 
		eY10102_Stn02UltrasonicGeneratorLeftRightOnOff                      	    :=19, 
		eY10103_Stn02UltrasonicGeneratorBottomOnOff                         	    :=20, 
		eY10104_Stn03UltrasonicGeneratorLeftRightOnOff                    	 	    :=21, 
		eY10105_Stn03UltrasonicGeneratorBottomOnOff                          	    :=22, 
		eY10106_Stn04UltrasonicGeneratorLeftRightOnOff                         	    :=23, 
		eY10107_Stn04UltrasonicGeneratorBottomOnOff                          	    :=24, 
		eY10108_Stn05UltrasonicGeneratorBottomOnOff                          	    :=25, 
		eY10109_Stn01DosingPumpOnOff                                              	:=26, 
		eY10110_Stn02DosingPumpOnOff                                              	:=27, 
		eY10111_Stn01ProcessTankPumpOnOff                                         	:=28, 
		eY10112_Stn02ProcessTankPumpOnOff                                         	:=29, 
		eY10113_Stn03ProcessTankPumpOnOff                                         	:=30, 
		eY10114_Stn04ProcessTankPumpOnOff                                         	:=31, 
		eY10115_Stn05ProcessTankPumpOnOff                                         	:=32, 
		                                                                          	       
		eY10200_Stn01_04ChemicalReturnTankPumpOnOff                               	:=33, 
		eY10201_Stn06ProcessTankVacuumPumpOnOff                                   	:=34, 
		eY10202_Stn01ProcessTankHeaterOnOff                                       	:=35, 
		eY10203_Stn02ProcessTankHeaterOnOff                                       	:=36, 
		eY10204_Stn03ProcessTankHeaterOnOff                                       	:=37, 
		eY10205_Stn04ProcessTankHeaterOnOff                                       	:=38, 
		eY10206_Stn06ProcessTankHeaterOnOff                                       	:=39, 
		eY10207_Stn06ProcessTankBlowerOnOff                                       	:=40, 
		eY10208_Stn01_06ExhaustBlowerOnOff                                        	:=41, 
		eY10209_Reserved                                                            :=42, 
		eY10210_Reserved                                                            :=43, 
		eY10211_Reserved                                                            :=44, 
		eY10212_Reserved                                                            :=45, 
		eY10213_Reserved                                                            :=46, 
		eY10214_Reserved                                                            :=47, 
		eY10215_Reserved                                                            :=48, 
		                                                                                  
		eY10300_Stn01_05AgitationMotorOnOff                                         :=49, 
		eY10301_LoadingConveyor01OnOff                                              :=50, 
		eY10302_LoadingConveyor02OnOff                                              :=51, 
		eY10303_LoadingConveyor03OnOff                                              :=52, 
		eY10304_StationRotationForRotaryBarrelOnOff                                 :=53, 
		eY10305_RobotRotationForRotaryBarrelOnOff                                   :=54, 
		eY10306_Reserved                                                            :=55, 
		eY10307_Reserved                                                            :=56, 
		eY10308_Reserved                                                            :=57, 
		eY10309_Reserved                                                            :=58, 
		eY10310_Reserved                                                            :=59, 
		eY10311_Reserved                                                            :=60, 
		eY10312_Reserved                                                            :=61, 
		eY10313_Reserved                                                            :=62, 
		eY10314_Reserved                                                            :=63, 
		eY10315_Reserved                                                            :=64, 
		                                                                                  
		eY11000_Stn03DosingPumpOnOff                                                :=65, 
		eY11001_Stn04DosingPumpOnOff                                                :=66, 
		eY11002_Reserved                                                            :=67, 
		eY11003_Reserved                                                            :=68, 
		eY11004_Reserved                                                            :=69, 
		eY11005_Reserved                                                            :=70, 
		eY11006_Reserved                                                            :=71, 
		eY11007_Reserved                                                            :=72, 
		eY11008_Reserved                                                            :=73, 
		eY11009_Reserved                                                            :=74, 
		eY11010_Reserved                                                            :=75, 
		eY11011_Reserved                                                            :=76, 
		eY11012_Reserved                                                            :=77, 
		eY11013_Reserved                                                            :=78, 
		eY11014_Reserved                                                            :=79, 
		eY11015_Reserved                                                            :=80, 
		                                                                                  
		eY12000_Stn01IncomingDiwSupplyAv1_1                                         :=81, 
		eY12001_Stn01OverflowSuctionAv1_2                                           :=82, 
		eY12002_Stn01BottomSuctionAv1_3                                             :=83, 
		eY12003_Stn01DrainAv1_4                                                     :=84, 
		eY12004_Stn02IncomingDiwSupplyAv2_1                                         :=85, 
		eY12005_Stn02OverflowSuctionAv2_2                                           :=86, 
		eY12006_Stn02BottomSuctionAv2_3                                             :=87, 
		eY12007_Stn02DrainAv2_4                                                     :=88, 
		eY12008_Stn03IncomingDiwSupplyAv3_1                                         :=89, 
		eY12009_Stn03OverflowSuctionAv3_2                                           :=90, 
		eY12010_Stn03BottomSuctionAv3_3                                             :=91, 
		eY12011_Stn03DrainAv3_4                                                     :=92, 
		eY12012_Stn04IncomingDiwSupplyAv4_1                                         :=93, 
		eY12013_Stn04OverflowSuctionAv4_2                                           :=94, 
		eY12014_Stn04BottomSuctionAv4_3                                             :=95, 
		eY12015_Stn04DrainAv4_4                                                     :=96, 
		                                                                                  
		eY12100_Stn05IncomingDiwSupplyAv5_1                                         :=97, 
		eY12101_Stn05IncomingCwSupplyAv5_2                                           :=98, 
		eY12102_Stn05BottomSuctionAv5_3                                             :=99, 
		eY12103_Stn05DrainAv5_4                                                     :=100,
		eY12104_Stn06BlowerProtectionAv6_1                                          :=101,
		eY12105_Stn06BlowerProtectionAv6_2                                          :=102,
		eY12106_Stn06VacuumSuctionAv6_3                                             :=103,
		eY12107_Stn06VacuumReleaseAv6_4                                             :=104,
		eY12108_GeneralIncomingDiwSupplyAvinc_1                                     :=105,
		eY12109_GeneralIncomingCwSupplyAvinc_2                                      :=106,
		eY12110_Reserved                                                            :=107,
		eY12111_Reserved                                                            :=108,
		eY12112_Reserved                                                            :=109,
		eY12113_Reserved                                                            :=110,
		eY12114_Reserved                                                            :=111,
		eY12115_Reserved                                                            :=112,
		                                                                                  
		eY12200_Stn06SlidingDoor_Open                                               :=113,
		eY12201_Stn06SlidingDoor_Close                                              :=114,
		eY12202_Stn06SlidingDoor_Clamp                                              :=115,
		eY12203_Stn06SlidingDoor_Unclamp                                            :=116,
		eY12204_Reserved                                                            :=117,
		eY12205_Reserved                                                            :=118,
		eY12206_Reserved                                                            :=119,
		eY12207_Reserved                                                            :=120,
		eY12208_Reserved                                                            :=121,
		eY12209_Reserved                                                            :=122,
		eY12210_Reserved                                                            :=123,
		eY12211_Reserved                                                            :=124,
		eY12212_Reserved                                                            :=125,
		eY12213_Reserved                                                            :=126,
		eY12214_Reserved                                                            :=127,
		eY12215_Reserved                                                            :=128

);
END_TYPE

// ---- DUTs/DS Twincat 3/Enum/Enum_Alarm_Others.TcDUT
{attribute 'Tc2GvlVarNames'}
{attribute 'strict'}
{attribute 'to_String'}

TYPE Enum_Alarm_Others :
(
			Stn01ProcessTankHighTempAlarm								:= 300,
			Stn02ProcessTankHighTempAlarm                               := 301,
			Stn03ProcessTankHighTempAlarm                               := 302,
			Stn04ProcessTankHighTempAlarm                               := 303,
			Stn05ProcessTankHighTempAlarm                               := 304,
			Stn06ProcessTankHighTempAlarm                               := 305,
			Stn07ProcessTankHighTempAlarm                               := 306,
			Stn08ProcessTankHighTempAlarm                               := 307,
			Stn09ProcessTankHighTempAlarm                               := 308,
			Stn10ProcessTankHighTempAlarm                               := 309,
			ProcessTank1TempPreparationNoReadyAlarm                     := 315,
			ProcessTank2TempPreparationNoReadyAlarm                     := 316,
			ProcessTank3TempPreparationNoReadyAlarm                     := 317,
			ProcessTank4TempPreparationNoReadyAlarm                     := 318,
			ProcessTank5TempPreparationNoReadyAlarm                     := 319,
			ProcessTank6TempPreparationNoReadyAlarm                     := 320,
			ProcessTank7TempPreparationNoReadyAlarm                     := 321,
			ProcessTank8TempPreparationNoReadyAlarm                     := 322,
			ProcessTank9TempPreparationNoReadyAlarm                     := 323,
			ProcessTank1TempOver1StLimitAlarm                           := 330,
			ProcessTank2TempOver1StLimitAlarm                           := 331,
			ProcessTank3TempOver1StLimitAlarm                           := 332,
			ProcessTank4TempOver1StLimitAlarm                           := 333,
			ProcessTank5TempOver1StLimitAlarm                           := 334,
			ProcessTank6TempOver1StLimitAlarm                           := 335,
			ProcessTank7TempOver1StLimitAlarm                           := 336,
			ProcessTank8TempOver1StLimitAlarm                           := 337,
			ProcessTank9TempOver1StLimitAlarm                           := 338,
			ProcessTank10TempOver1StLimitAlarm                          := 339,
			ProcessTank1TempOver2NdLimitAlarm                           := 346,
			ProcessTank2TempOver2NdLimitAlarm                           := 347,
			ProcessTank3TempOver2NdLimitAlarm                           := 348,
			ProcessTank4TempOver2NdLimitAlarm                           := 349,
			ProcessTank5TempOver2NdLimitAlarm                           := 350,
			ProcessTank6TempOver2NdLimitAlarm                           := 351,
			ProcessTank7TempOver2NdLimitAlarm                           := 352,
			ProcessTank8TempOver2NdLimitAlarm                           := 353,
			ProcessTank9TempOver2NdLimitAlarm                           := 354,
			ProcessTank10TempOver2NdLimitAlarm                          := 355,
			ProcessTank11TempOver2NdLimitAlarm                          := 356,
			ProcessTank12TempOver2NdLimitAlarm                          := 357,
			IncTempOver2NdLimitAlarm                                    := 358,
			StnWaterJacketTempOver2NdLimitAlarm                         := 359,
			ProcessTank1ConductivityLowAlarm                            := 360,
			ProcessTank2ConductivityLowAlarm                            := 361,
			ProcessTank3ConductivityLowAlarm                            := 362,
			ProcessTank4ConductivityLowAlarm                            := 363,
			ProcessTank5ConductivityLowAlarm                            := 364,
			ProcessTank6ConductivityLowAlarm                            := 365,
			ProcessTank7ConductivityLowAlarm                            := 366,
			ProcessTank8ConductivityLowAlarm                            := 367,
			ProcessTank1PressureSwitchLowAlarm                          := 368,
			ProcessTank2PressureSwitchLowAlarm                          := 369,
			ProcessTank3PressureSwitchLowAlarm                          := 370,
			ProcessTank4PressureSwitchLowAlarm                          := 371,
			ProcessTank5PressureSwitchLowAlarm                          := 372,
			ProcessTank6PressureSwitchLowAlarm                          := 373,
			ProcessTank7PressureSwitchLowAlarm                          := 374,
			ProcessTank8PressureSwitchLowAlarm                          := 375,
			ProcessTank9PressureSwitchLowAlarm                          := 376,
			ProcessTank1ConductivityHighAlarm                           := 380,
			ProcessTank2ConductivityHighAlarm                           := 381,
			ProcessTank3ConductivityHighAlarm                           := 382,
			ProcessTank4ConductivityHighAlarm                           := 383,
			ProcessTank5ConductivityHighAlarm                           := 384,
			ProcessTank6ConductivityHighAlarm                           := 385,
			ProcessTank7ConductivityHighAlarm                           := 386,
			ProcessTank8ConductivityHighAlarm                           := 387,
			ProcessTank1PressureSwitchHighAlarm                         := 388,
			ProcessTank2PressureSwitchHighAlarm                         := 389,
			ProcessTank3PressureSwitchHighAlarm                         := 390,
			ProcessTank4PressureSwitchHighAlarm                         := 391,
			ProcessTank5PressureSwitchHighAlarm                         := 392,
			ProcessTank6PressureSwitchHighAlarm                         := 393,
			ProcessTank7PressureSwitchHighAlarm                         := 394,
			ProcessTank8PressureSwitchHighAlarm                         := 395,
			ProcessTank9PressureSwitchHighAlarm                         := 396,
			ProcessTank1BadBasket_OverToleranceTime                     := 400,
			ProcessTank2BadBasket_OverToleranceTime                     := 401,
			ProcessTank3BadBasket_OverToleranceTime                     := 402,
			ProcessTank4BadBasket_OverToleranceTime                     := 403,
			ProcessTank5BadBasket_OverToleranceTime                     := 404,
			ProcessTank6BadBasket_OverToleranceTime                     := 405,
			ProcessTank7BadBasket_OverToleranceTime                     := 406,
			ProcessTank8BadBasket_OverToleranceTime                     := 407,
			ProcessTank9BadBasket_OverToleranceTime                     := 408,
			ProcessTank10BadBasket_OverToleranceTime                    := 409,
			ProcessTank11BadBasket_OverToleranceTime                    := 410,
			ProcessTank12BadBasket_OverToleranceTime                    := 411,
			Arm1OvertimeError                                           := 412,
			Arm2OvertimeError                                           := 413,
			SlowpullLifterError                                         := 414,
			ProcessTank1DosingPumpHealthACheckPulseError                := 415,
			ProcessTank2DosingPumpHealthACheckPulseError                := 416,
			ProcessTank3DosingPumpHealthACheckPulseError                := 417,
			ProcessTank4DosingPumpHealthACheckPulseError				:= 418,
			Arm1VerticalUpOverTravelAlarm                               := 421,
			Arm1VerticalDownOverTravelAlarm                             := 422,
			Arm1VerticalErrorStopAlarm                                  := 423,
			Arm1HorizontalLoadingOverTravelAlarm                        := 424,
			Arm1HorizontalUnloadingOverTravelAlarm                      := 425,
			Arm1HorizontalErrorStopAlarm                                := 426,
			SlowpullUpOverTravelAlarm                                   := 427,
			SlowpullDownOverTravelAlarm                                 := 428,
			SlowpullErrorStopAlarm                                      := 429,
			DcPowerUnknownStatusAlarm                                   := 430,
			UpsCommUnknownStatusAlarm                                   := 431,
			BatteryReplacementRequestAlarm                              := 432,
			UpsCommErrorAlarm                                           := 433,
			Arm1VerticalAxisError                                       := 434,
			Arm1HorizontalAxisError                                     := 435,
			Arm2VerticalAxisError                                       := 436,
			Arm2HorizontalAxisError                                     := 437,
			MasterTimeBlockWriteArmDataError                            := 438,
			MasterTimeBlockWriteStnDataError                            := 439,
			MasterTimeBlockNoAvailableSlotError                         := 440,
			VacuumPumpRoutineServiceReminderAlarmReached				:= 441,
			VacuumPumpMajorWarningServiceReminder						:= 442,
			VacuumPumpMajorServiceReminderAlarmReached					:= 443,	
			LoadingCallArmSpeedProfileMemoryError                       := 444,
			LoadingCallPickStationNoError                               := 445,
			LoadingCallTransferStationNoError                           := 446,
			LoadingCallUpDownPatternMemoryError                         := 447,
			LoadingInvalidProductRecipeNoErrorHold                      := 448,
			LoadingInvalidProductRecipeStepErrorHold                    := 449,
			StationCallArmSpeedProfileMemoryError                       := 450,
			StationCallPickStationNoError                               := 451,
			StationCallTransferStationNoError                           := 452,
			StationCallUpDownPatternMemoryError                         := 453,
			StationInvalidProductRecipeNoErrorHold                      := 454,
			StationInvalidProductRecipeStepErrorHold                    := 455

);
END_TYPE

// ---- DUTs/DS Twincat 3/Event/DS_ActiveEventDisplay.TcDUT
TYPE DS_ActiveEventDisplay EXTENDS DS_EventDescriptionCausedRemedy :
STRUCT

	iEventID						: INT; (*To Keep the array number ot repersent as Event ID when it stored in Event logger*)
	sTimeAndDate_Occurred 			: STRING(50);

END_STRUCT
END_TYPE

// ---- DUTs/DS Twincat 3/Event/DS_Event.TcDUT
TYPE DS_Event :
STRUCT
	iEventID						: INT; (*To Keep the array number ot repersent as Event ID when it stored in Event logger*)
	sTimeAndDate_Occurred 			: STRING(50);
	
END_STRUCT
END_TYPE

// ---- DUTs/DS Twincat 3/Event/DS_EventControl.TcDUT
TYPE DS_EventControl :
STRUCT
	bSignalInput 					: BOOL;
	bHoldingDisable 				: BOOL;
	bTest_InvertedInputEn			: BOOL;
	eEventType						: E_EventType;
	iDelayTimeSV					: INT;
	iDelayTimeEV					: INT;
	bEventOutput					: BOOL;
	bEventBuzzerStop				: BOOL;
	
END_STRUCT
END_TYPE

// ---- DUTs/DS Twincat 3/Event/DS_EventDescriptionCausedRemedy.TcDUT
TYPE DS_EventDescriptionCausedRemedy :
STRUCT
	sEventCode						: STRING(10);
	sEventType						: STRING(10);
	sLocation						: STRING(20);
	sSubLocation					: STRING(20);
	sDescription 					: STRING(80);
	sCaused							: STRING(80);
	sRemedy							: STRING(220);

END_STRUCT
END_TYPE

// ---- DUTs/DS Twincat 3/Event/DS_EventHistory.TcDUT
TYPE DS_EventHistory EXTENDS DS_Event :
STRUCT
	sTimeAndDate_Recovered 			: STRING(50);
	sTimeAndDate_Acknowledged 		: STRING(50);
	
END_STRUCT
END_TYPE

// ---- DUTs/DS Twincat 3/Event/DS_EventHistoryLogToFile.TcDUT
TYPE DS_EventHistoryLogToFile EXTENDS DS_EventHistory :
STRUCT
	sEventCode						: STRING(10);
	sEventType						: STRING(10);
	sLocation						: STRING(20);
	sSubLocation					: STRING(20);
	sDescription 					: STRING(80);
END_STRUCT
END_TYPE

// ---- DUTs/DS Twincat 3/Event/DS_HistoryEventDisplay.TcDUT
TYPE DS_HistoryEventDisplay EXTENDS DS_EventDescriptionCausedRemedy :
STRUCT
	
	iEventID						: INT; (*To Keep the array number ot repersent as Event ID when it stored in Event logger*)
	sTimeAndDate_Occurred 			: STRING(50);
	sTimeAndDate_Recovered 			: STRING(50);
	sTimeAndDate_Acknowledged 		: STRING(50);

END_STRUCT
END_TYPE

// ---- DUTs/DS Twincat 3/Event/E_EventType.TcDUT
{attribute 'qualified_only'}
{attribute 'strict'}
{attribute 'to_string'}
TYPE E_EventType :
(
	Caution := 0,
	Warning := 1,
	Error	:= 2

);
END_TYPE

// ---- DUTs/DS Twincat 3/E_HmiLanguage.TcDUT
{attribute 'qualified_only'}
{attribute 'strict'}
TYPE E_HmiLanguage :
(
	English 	:= 1,
	Mandarin 	:= 2,
	German 		:= 3,
	French 		:= 4,
	Portuguese 	:= 5
);
END_TYPE

// ---- DUTs/DS Twincat 3/ST_DataLog.TcDUT
TYPE ST_DataLog :
STRUCT
	sName:STRING;
	sName1:STRING;
	sName2:STRING;
	sName3:STRING;
	sName4:STRING;
	sValue:STRING;
END_STRUCT
END_TYPE

// ---- DUTs/DS Twincat 3/UserCtrl/DS_HmiUserReg.TcDUT
TYPE DS_HmiUserReg :
STRUCT 
	ARsOperatorIdentifier	: ARRAY [0..20+1] OF STRING;	// Celestica Requirement	
	AReActorType			: ARRAY [0..20+1] OF eActor;	// Celestica Requirement
	ARsLastName				: ARRAY [0..20+1] OF STRING;
	ARsFirstName 			: ARRAY [0..20+1] OF STRING;
	ARsLoginName			: ARRAY [0..20+1] OF STRING;	// Same as Username
	ARbUserStatus			: ARRAY [0..20+1] OF BOOL; 	// 0 = Deactivated/Disable, 1 = Active User
	
	ARiUserGroupID			: ARRAY [0..20+1] OF INT; 	// Define in HMI TF1800
	ARwsUserGroupName		: ARRAY [0..20+1] OF WSTRING; 	// Define in HMI TF1800
	ARsPw					: ARRAY [0..20+1] OF STRING;
	
	iQtyUserReg				: INT := 20;

END_STRUCT

END_TYPE

// ---- DUTs/DS Twincat 3/UserCtrl/DS_HmiUserStatus.TcDUT
TYPE DS_HmiUserStatus :
STRUCT
	
	bActivatedFlag 		: BOOL;
	sLoginName			: STRING;	// User Management - New User Login Name
	sUserGroupId		: INT;		// User Management - Select from UserGroupList

	sOperatorIdentifier	: STRING;
	eActorType			: eActor;
	sULastName			: STRING;
	sFirstName			: STRING;	
	tsDateTime			: TIMESTRUCT;
	
	
END_STRUCT
END_TYPE

// ---- DUTs/DS Twincat 3/UserCtrl/DS_VisuElement.TcDUT
TYPE DS_VisuElement :
STRUCT
	CurrentUserGroupId 	: int;
	CurrentUserName		: WSTRING;
	CurrentVisu			: STRING;

	
END_STRUCT
END_TYPE

// ---- DUTs/DS Twincat 3/UserCtrl/eActorType.TcTLEO
{attribute 'qualified_only'}
{attribute 'strict'}
TYPE eActor :
(
	Human 			:= 0,
	Robot			:= 1,
	RemoteSystem	:= 2
);
END_TYPE

// ---- DUTs/DS Twincat 3/XML/E_XmlParType.TcDUT
{attribute 'Tc2GvlVarNames'}
{attribute 'strict'}
TYPE E_XmlParType :
(
	eXmlParTypeProductRecipe := 1,
	eXmlParTypeSSER := 2,
	eXmlParTypeSSUR := 3,
	eXmlParTypeSSMR := 4
);
END_TYPE

// ---- DUTs/DS Twincat 3/XML/E_XmlRwMode.TcDUT
{attribute 'Tc2GvlVarNames'}
{attribute 'strict'}
TYPE E_XmlRwMode :
(
	eXmlMode_MergeAllByType 					:= 1,			// SSER -> One XML, SSUR -> One XML, Product Recipe -> One XML and so on
	eXmlMode_SeperateByProductAndStation		:= 2,			// SSER will seperate by Station with Multiple file, same goes to the rest of the Recipe
	eXmlMode_SeperateAll					 	:= 3			// Seperate each of the recipe individually


);
END_TYPE

// ---- DUTs/DS Twincat 3/XML/E_XmlVariableType.TcDUT
{attribute 'Tc2GvlVarNames'}
{attribute 'strict'}
TYPE E_XmlVariableType :
(
	eXmlSSMR := 1,
	eXmlSSUR := 2,
	eXmlSSER := 3,
	eXmlProductRecipe := 4
);
END_TYPE

// ---- GVLs/Alarm_Ctrl/Global_Variables_Alarm.TcGVL
{attribute 'Tc2GvlVarNames'}
VAR_GLOBAL PERSISTENT

	fbAlarmModule_Main									: fbAlarmModule;

(*Input*)

	ARbSignalInput 										: ARRAY [1..iAlarmQty] OF BOOL;
	ARiDelayTimeSV 										: ARRAY [1..iAlarmQty] OF INT;

	ARsAlarmDescription 									: ARRAY [0..iAlarmQty] OF STRING(99);
	ARbHoldingDisable 									: ARRAY [1..iAlarmQty] OF BOOL;
	ARsDeactivateDescription							 	: ARRAY [0..iDeactivateQty] OF STRING(99);

	ARbTestAlarmEn	 									: ARRAY [1..iAlarmQty] OF BOOL;
	ARbTestSignal	 									: ARRAY [1..iAlarmQty] OF BOOL;

	bAlarmDeactivated									: BOOL ;

(*Output*)

	ARiDelayTimeEV	 									: ARRAY [1..iAlarmQty] OF INT;
	ARbAlarmOutput 										: ARRAY [1..iAlarmQty] OF BOOL;
	ARbDeactivateOutput 									: ARRAY [1..iDeactivateQty] OF BOOL;

	ARsAlarmDisplay										: ARRAY [0..iActAlarmDisplayQty] OF STRING(99);
(*	ARsAlarmDisplayStorage								: ARRAY [0..iActAlarmDisplayStorageQty] OF STRING(99);*)
	ARsAlarmAddressStore								: ARRAY [0..iActAlarmDisplayStorageQty] OF INT;

	ARsLoggingAlarmDisplay								: ARRAY [0..iLogAlarmDisplayQty] OF STRING(99);
	ARsLoggingOcrTimeDisplay							: ARRAY [0..iLogAlarmDisplayQty] OF STRING(99);
	ARsLoggingRcvTimeDisplay							: ARRAY [0..iLogAlarmDisplayQty] OF STRING(99);

	ARbArmOvertimeError									: ARRAY [1..iArmQty] OF BOOL;

	bAlarmOccurFlag										: BOOL;
	bBuzzerOccur											: BOOL ;

	ARbArmLifterError										: ARRAY [1..iArmSlowPullQty] OF BOOL;
	ARbArmLifterDriveErr									: ARRAY [1..iArmSlowPullQty] OF BOOL;
	ARbArmLifterAlarm									: ARRAY [1..iArmSlowPullQty] OF BOOL;

END_VAR

// ---- GVLs/Analog_Ctrl/Global_Variables_Analog_NoPersistent.TcGVL
{attribute 'Tc2GvlVarNames'}
VAR_GLOBAL

(* xxxxxxxxxxxxxxxxxxxxxxxxxxxxxxxx Temperature Cltr xxxxxxxxxxxxxxxxxxxxxxxxxxxxxxxx*)
(*========================================================================*)

	ARrStnTempPV										: ARRAY [1..iStnQty] OF REAL;
	ARbStnTempOnOff										: ARRAY [1..iStnQty] OF BOOL;
	ARbStnTempRDY										: ARRAY [1..iStnQty] OF BOOL;
	ARbStnTempHAL										: ARRAY [1..iStnQty] OF BOOL;
	ARbStnTemp1stLimitAlarm								: ARRAY [1..iStnQty] OF BOOL;
	ARbStnTemp2ndLimitAlarm								: ARRAY [1..iStnQty] OF BOOL;
	ARbStnTempPreparationNoRdyAlarm						: ARRAY [1..iStnQty] OF BOOL;

	rStnTempMINsvHMIDisplay								: REAL;
	rStnTempMAXsvHMIDisplay								: REAL;
	
	rStnTempHALMINsvHMIDisplay							: REAL;
	rStnTempHALMAXsvHMIDisplay							: REAL;
	
	rStnTempHYSMINsvHMIDisplay							: REAL;
	rStnTempHYSMAXsvHMIDisplay							: REAL;
	
	rStnTempRDYMINsvHMIDisplay							: REAL;
	rStnTempRDYMAXsvHMIDisplay							: REAL;
	
	rStnTemp1stLimitMINsvHMIDisplay						: REAL;
	rStnTemp1stLimitMAXsvHMIDisplay						: REAL;
	
	iStnPreparationTempMINsvHMIDisplay					: INT;
	iStnPreparationTempMAXsvHMIDisplay					: INT;	
	
	rChillerSystemTempPV								: REAL;
	bChillerSystemTempOnOff								: BOOL;
	bChillerSystemTempRDY								: BOOL;
	bChillerSystemTempHAL								: BOOL;
	bChillerSystemTemp1stLimitAlarm						: BOOL;
	bChillerSystemTemp2ndLimitAlarm						: BOOL;
	bChillerSystemTempPreparationNoRdyAlarm				: BOOL;
	
	ARbStnChillerValueOnOff								: ARRAY [1..iStnQty] OF BOOL;
	
(*****Temperature Changed Based on Recipe Ctrl *****)

	bDefaultTempSettingOnTSpagePB						: BOOL;
	iHMIrecipeFinalDestination							: INT;
	iCallProductRecipeFinalDestination					: INT;

	Call_bCallPB										: BOOL;

	bCallCompleted 										: BOOL;
	bInvalidCallTempCtrlRecipeHold						: BOOL;
	bInvalidCallTempCtrlRecipePulse						: BOOL;
	Call_DSTempCtrlRecipe 								: DSV3_TempCtrlRecipe;

(* xxxxxxxxxxxxxxxxxxxxxxxxxxxxxxxx Conductivity Cltr xxxxxxxxxxxxxxxxxxxxxxxxxxxxxxxx*)
(*========================================================================*)

	ARrStnConductivityPV 								: ARRAY [1..iStnQty] OF REAL;
	ARbStnConductivity1stLimitAlarm						: ARRAY [1..iStnQty] OF BOOL;
	ARbStnConductivity2ndLimitAlarm						: ARRAY [1..iStnQty] OF BOOL;
	
	ARbStnConductivityLowAlarm							: ARRAY [1..iStnQty] OF BOOL;
	ARbStnConductivityHighAlarm							: ARRAY [1..iStnQty] OF BOOL;
	
	ARtDelayOffTopupBasedConductivityTimerOn			: ARRAY [0..iStnQty] OF TON;

(* xxxxxxxxxxxxxxxxxxxxxxxxxxxxxxxx Resistivity Cltr xxxxxxxxxxxxxxxxxxxxxxxxxxxxxxxx*)
(*========================================================================*)

	ARrStnResistivityPV 									: ARRAY [1..iStnQty] OF REAL;
	ARbStnResistivity1stLimitAlarm							: ARRAY [1..iStnQty] OF BOOL;
	ARbStnResistivity2ndLimitAlarm							: ARRAY [1..iStnQty] OF BOOL;

	rIncResistivityPV 										: REAL;
	bIncResistivity1stLimitAlarm							: BOOL;
	bIncResistivity2ndLimitAlarm							: BOOL;

(* xxxxxxxxxxxxxxxxxxxxxxxxxxxxxxxx PH Cltr xxxxxxxxxxxxxxxxxxxxxxxxxxxxxxxx*)
(*========================================================================*)

	ARrStnPhPV 											: ARRAY [1..iStnQty] OF REAL;
	ARbStnPH1stLimitAlarm								: ARRAY [1..iStnQty] OF BOOL;
	ARbStnPH2ndLimitAlarm								: ARRAY [1..iStnQty] OF BOOL;

(* xxxxxxxxxxxxxxxxxxxxxxxxxxxxxxxx Filter Pressure Cltr xxxxxxxxxxxxxxxxxxxxxxxxxxxxxxxx*)
(*========================================================================*)

